    movel([0.140497, -1.371488, -2.576513, -0.764389, 1.570796, 1.711294],accel_mss,speed_ms,0,blend_radius_m)
    movel([0.140657, -1.371181, -2.576725, -0.764483, 1.570796, 1.711454],accel_mss,speed_ms,0,blend_radius_m)
    movel([0.140844, -1.370889, -2.576927, -0.764572, 1.570796, 1.711640],accel_mss,speed_ms,0,blend_radius_m)
    movel([0.141059, -1.370603, -2.577125, -0.764661, 1.570796, 1.711855],accel_mss,speed_ms,0,blend_radius_m)
    movel([0.141302, -1.370327, -2.577316, -0.764746, 1.570796, 1.712098],accel_mss,speed_ms,0,blend_radius_m)
    movel([0.141561, -1.370068, -2.577495, -0.764826, 1.570796, 1.712357],accel_mss,speed_ms,0,blend_radius_m)
    movel([0.141844, -1.369824, -2.577664, -0.764901, 1.570796, 1.712640],accel_mss,speed_ms,0,blend_radius_m)
    movel([0.142141, -1.369603, -2.577817, -0.764969, 1.570796, 1.712937],accel_mss,speed_ms,0,blend_radius_m)
    movel([0.142479, -1.369380, -2.577971, -0.765038, 1.570796, 1.713275],accel_mss,speed_ms,0,blend_radius_m)
    movel([0.142834, -1.369176, -2.578112, -0.765102, 1.570796, 1.713630],accel_mss,speed_ms,0,blend_radius_m)
    movel([0.143191, -1.368999, -2.578233, -0.765156, 1.570796, 1.713987],accel_mss,speed_ms,0,blend_radius_m)
    movel([0.143557, -1.368846, -2.578339, -0.765204, 1.570796, 1.714353],accel_mss,speed_ms,0,blend_radius_m)
    movel([0.143920, -1.368724, -2.578423, -0.765242, 1.570796, 1.714717],accel_mss,speed_ms,0,blend_radius_m)
    movel([0.144279, -1.368628, -2.578489, -0.765272, 1.570796, 1.715076],accel_mss,speed_ms,0,blend_radius_m)
    movel([0.144633, -1.368564, -2.578533, -0.765292, 1.570796, 1.715430],accel_mss,speed_ms,0,blend_radius_m)
    movel([0.144980, -1.368530, -2.578557, -0.765302, 1.570796, 1.715776],accel_mss,speed_ms,0,blend_radius_m)
    movel([0.145312, -1.368525, -2.578561, -0.765304, 1.570796, 1.716108],accel_mss,speed_ms,0,blend_radius_m)
    movel([0.145619, -1.368551, -2.578542, -0.765296, 1.570796, 1.716416],accel_mss,speed_ms,0,blend_radius_m)
    movel([0.145910, -1.368604, -2.578506, -0.765279, 1.570796, 1.716707],accel_mss,speed_ms,0,blend_radius_m)
    movel([0.146159, -1.368679, -2.578454, -0.765256, 1.570796, 1.716955],accel_mss,speed_ms,0,blend_radius_m)
    movel([0.146381, -1.368783, -2.578382, -0.765223, 1.570796, 1.717177],accel_mss,speed_ms,0,blend_radius_m)
    movel([0.146581, -1.368916, -2.578291, -0.765182, 1.570796, 1.717377],accel_mss,speed_ms,0,blend_radius_m)
    movel([0.146755, -1.369074, -2.578182, -0.765133, 1.570796, 1.717551],accel_mss,speed_ms,0,blend_radius_m)
    movel([0.146898, -1.369260, -2.578054, -0.765076, 1.570796, 1.717694],accel_mss,speed_ms,0,blend_radius_m)
    movel([0.147008, -1.369466, -2.577911, -0.765012, 1.570796, 1.717805],accel_mss,speed_ms,0,blend_radius_m)
    movel([0.147132, -1.369810, -2.577674, -0.764905, 1.570796, 1.717928],accel_mss,speed_ms,0,blend_radius_m)
    movel([0.147248, -1.370196, -2.577407, -0.764786, 1.570796, 1.718044],accel_mss,speed_ms,0,blend_radius_m)
    movel([0.147260, -1.370511, -2.577189, -0.764689, 1.570796, 1.718057],accel_mss,speed_ms,0,blend_radius_m)
    movel([0.147149, -1.370874, -2.576938, -0.764577, 1.570796, 1.717945],accel_mss,speed_ms,0,blend_radius_m)
    movel([0.146700, -1.371702, -2.576364, -0.764323, 1.570796, 1.717496],accel_mss,speed_ms,0,blend_radius_m)
    movel([0.146700, -1.374505, -2.577635, -0.760249, 1.570796, 1.717496],accel_mss,speed_ms,0,blend_radius_m)
    movel([0.146515, -1.374803, -2.577427, -0.760159, 1.570796, 1.717312],accel_mss,speed_ms,0,blend_radius_m)
    movel([0.146310, -1.375097, -2.577222, -0.760070, 1.570796, 1.717106],accel_mss,speed_ms,0,blend_radius_m)
    movel([0.146072, -1.375395, -2.577014, -0.759980, 1.570796, 1.716868],accel_mss,speed_ms,0,blend_radius_m)
    movel([0.145854, -1.375635, -2.576846, -0.759907, 1.570796, 1.716651],accel_mss,speed_ms,0,blend_radius_m)
    movel([0.145623, -1.375855, -2.576693, -0.759841, 1.570796, 1.716419],accel_mss,speed_ms,0,blend_radius_m)
    movel([0.145375, -1.376060, -2.576550, -0.759779, 1.570796, 1.716171],accel_mss,speed_ms,0,blend_radius_m)
    movel([0.145105, -1.376251, -2.576416, -0.759722, 1.570796, 1.715901],accel_mss,speed_ms,0,blend_radius_m)
    movel([0.144824, -1.376424, -2.576295, -0.759670, 1.570796, 1.715620],accel_mss,speed_ms,0,blend_radius_m)
    movel([0.144503, -1.376590, -2.576180, -0.759620, 1.570796, 1.715300],accel_mss,speed_ms,0,blend_radius_m)
    movel([0.144154, -1.376739, -2.576075, -0.759575, 1.570796, 1.714951],accel_mss,speed_ms,0,blend_radius_m)
    movel([0.143741, -1.376887, -2.575972, -0.759531, 1.570796, 1.714537],accel_mss,speed_ms,0,blend_radius_m)
    movel([0.143329, -1.377009, -2.575886, -0.759494, 1.570796, 1.714125],accel_mss,speed_ms,0,blend_radius_m)
    movel([0.142981, -1.377092, -2.575828, -0.759469, 1.570796, 1.713778],accel_mss,speed_ms,0,blend_radius_m)
    movel([0.142643, -1.377148, -2.575789, -0.759452, 1.570796, 1.713439],accel_mss,speed_ms,0,blend_radius_m)
    movel([0.142311, -1.377177, -2.575769, -0.759444, 1.570796, 1.713108],accel_mss,speed_ms,0,blend_radius_m)
    movel([0.141991, -1.377179, -2.575767, -0.759443, 1.570796, 1.712788],accel_mss,speed_ms,0,blend_radius_m)
    movel([0.141699, -1.377158, -2.575782, -0.759449, 1.570796, 1.712495],accel_mss,speed_ms,0,blend_radius_m)
    movel([0.141435, -1.377113, -2.575813, -0.759463, 1.570796, 1.712231],accel_mss,speed_ms,0,blend_radius_m)
    movel([0.141198, -1.377045, -2.575861, -0.759483, 1.570796, 1.711994],accel_mss,speed_ms,0,blend_radius_m)
    movel([0.140980, -1.376950, -2.575927, -0.759512, 1.570796, 1.711776],accel_mss,speed_ms,0,blend_radius_m)
    movel([0.140781, -1.376828, -2.576013, -0.759548, 1.570796, 1.711577],accel_mss,speed_ms,0,blend_radius_m)
    movel([0.140605, -1.376681, -2.576115, -0.759592, 1.570796, 1.711401],accel_mss,speed_ms,0,blend_radius_m)
    movel([0.140456, -1.376512, -2.576233, -0.759643, 1.570796, 1.711253],accel_mss,speed_ms,0,blend_radius_m)
    movel([0.140339, -1.376327, -2.576363, -0.759699, 1.570796, 1.711135],accel_mss,speed_ms,0,blend_radius_m)
    movel([0.140254, -1.376124, -2.576505, -0.759760, 1.570796, 1.711050],accel_mss,speed_ms,0,blend_radius_m)
    movel([0.140198, -1.375902, -2.576660, -0.759827, 1.570796, 1.710994],accel_mss,speed_ms,0,blend_radius_m)
    movel([0.140172, -1.375669, -2.576823, -0.759897, 1.570796, 1.710969],accel_mss,speed_ms,0,blend_radius_m)
    movel([0.140176, -1.375422, -2.576995, -0.759972, 1.570796, 1.710972],accel_mss,speed_ms,0,blend_radius_m)
    movel([0.140213, -1.375145, -2.577188, -0.760055, 1.570796, 1.711009],accel_mss,speed_ms,0,blend_radius_m)
    movel([0.140277, -1.374866, -2.577383, -0.760140, 1.570796, 1.711073],accel_mss,speed_ms,0,blend_radius_m)
    movel([0.140374, -1.374578, -2.577583, -0.760227, 1.570796, 1.711170],accel_mss,speed_ms,0,blend_radius_m)
    movel([0.140497, -1.374290, -2.577784, -0.760315, 1.570796, 1.711294],accel_mss,speed_ms,0,blend_radius_m)
    movel([0.140657, -1.373985, -2.577997, -0.760407, 1.570796, 1.711454],accel_mss,speed_ms,0,blend_radius_m)
    movel([0.140844, -1.373694, -2.578199, -0.760496, 1.570796, 1.711640],accel_mss,speed_ms,0,blend_radius_m)
    movel([0.141059, -1.373408, -2.578398, -0.760583, 1.570796, 1.711855],accel_mss,speed_ms,0,blend_radius_m)
    movel([0.141302, -1.373132, -2.578589, -0.760667, 1.570796, 1.712098],accel_mss,speed_ms,0,blend_radius_m)
    movel([0.141561, -1.372874, -2.578769, -0.760746, 1.570796, 1.712357],accel_mss,speed_ms,0,blend_radius_m)
    movel([0.141844, -1.372631, -2.578938, -0.760821, 1.570796, 1.712640],accel_mss,speed_ms,0,blend_radius_m)
    movel([0.142141, -1.372410, -2.579091, -0.760888, 1.570796, 1.712937],accel_mss,speed_ms,0,blend_radius_m)
    movel([0.142479, -1.372187, -2.579245, -0.760957, 1.570796, 1.713275],accel_mss,speed_ms,0,blend_radius_m)
    movel([0.142834, -1.371984, -2.579386, -0.761019, 1.570796, 1.713630],accel_mss,speed_ms,0,blend_radius_m)
    movel([0.143191, -1.371807, -2.579508, -0.761073, 1.570796, 1.713987],accel_mss,speed_ms,0,blend_radius_m)
    movel([0.143557, -1.371655, -2.579614, -0.761120, 1.570796, 1.714353],accel_mss,speed_ms,0,blend_radius_m)
    movel([0.143920, -1.371533, -2.579699, -0.761158, 1.570796, 1.714717],accel_mss,speed_ms,0,blend_radius_m)
    movel([0.144279, -1.371437, -2.579765, -0.761187, 1.570796, 1.715076],accel_mss,speed_ms,0,blend_radius_m)
    movel([0.144633, -1.371373, -2.579809, -0.761207, 1.570796, 1.715430],accel_mss,speed_ms,0,blend_radius_m)
    movel([0.144980, -1.371339, -2.579833, -0.761217, 1.570796, 1.715776],accel_mss,speed_ms,0,blend_radius_m)
    movel([0.145312, -1.371334, -2.579836, -0.761219, 1.570796, 1.716108],accel_mss,speed_ms,0,blend_radius_m)
    movel([0.145619, -1.371361, -2.579818, -0.761211, 1.570796, 1.716416],accel_mss,speed_ms,0,blend_radius_m)
    movel([0.145910, -1.371413, -2.579782, -0.761195, 1.570796, 1.716707],accel_mss,speed_ms,0,blend_radius_m)
    movel([0.146159, -1.371489, -2.579729, -0.761171, 1.570796, 1.716955],accel_mss,speed_ms,0,blend_radius_m)
    movel([0.146381, -1.371592, -2.579658, -0.761139, 1.570796, 1.717177],accel_mss,speed_ms,0,blend_radius_m)
    movel([0.146581, -1.371724, -2.579566, -0.761099, 1.570796, 1.717377],accel_mss,speed_ms,0,blend_radius_m)
    movel([0.146755, -1.371882, -2.579456, -0.761050, 1.570796, 1.717551],accel_mss,speed_ms,0,blend_radius_m)
    movel([0.146898, -1.372067, -2.579328, -0.760993, 1.570796, 1.717694],accel_mss,speed_ms,0,blend_radius_m)
    movel([0.147008, -1.372273, -2.579186, -0.760930, 1.570796, 1.717805],accel_mss,speed_ms,0,blend_radius_m)
    movel([0.147132, -1.372616, -2.578948, -0.760825, 1.570796, 1.717928],accel_mss,speed_ms,0,blend_radius_m)
    movel([0.147248, -1.373001, -2.578680, -0.760707, 1.570796, 1.718044],accel_mss,speed_ms,0,blend_radius_m)
    movel([0.147260, -1.373316, -2.578462, -0.760611, 1.570796, 1.718057],accel_mss,speed_ms,0,blend_radius_m)
    movel([0.147149, -1.373678, -2.578210, -0.760501, 1.570796, 1.717945],accel_mss,speed_ms,0,blend_radius_m)
    movel([0.146700, -1.374505, -2.577635, -0.760249, 1.570796, 1.717496],accel_mss,speed_ms,0,blend_radius_m)
    movel([0.146700, -1.341961, -2.561990, -0.808439, 1.570796, 1.717496],accel_mss,speed_ms,0,blend_radius_m)
    speed_ms = 1.000
    movel([0.156390, -1.339995, -2.563292, -0.809102, 1.570796, 1.727187],accel_mss,speed_ms,0,blend_radius_m)
    speed_ms = 0.008
    movel([0.156390, -1.366441, -2.576163, -0.769785, 1.570796, 1.727187],accel_mss,speed_ms,0,blend_radius_m)
    speed_ms = 0.003
    movel([0.156390, -1.369779, -2.577695, -0.764915, 1.570796, 1.727187],accel_mss,speed_ms,0,blend_radius_m)
    speed_ms = 0.008
    movel([0.155185, -1.370065, -2.577497, -0.764827, 1.570796, 1.725981],accel_mss,speed_ms,0,blend_radius_m)
    movel([0.156709, -1.361432, -2.583412, -0.767545, 1.570796, 1.727505],accel_mss,speed_ms,0,blend_radius_m)
    movel([0.159145, -1.360847, -2.583810, -0.767733, 1.570796, 1.729942],accel_mss,speed_ms,0,blend_radius_m)
    movel([0.157596, -1.369493, -2.577893, -0.765003, 1.570796, 1.728393],accel_mss,speed_ms,0,blend_radius_m)
    movel([0.156390, -1.369779, -2.577695, -0.764915, 1.570796, 1.727187],accel_mss,speed_ms,0,blend_radius_m)
    movel([0.156390, -1.372585, -2.578969, -0.760835, 1.570796, 1.727187],accel_mss,speed_ms,0,blend_radius_m)
    movel([0.155185, -1.372871, -2.578771, -0.760747, 1.570796, 1.725981],accel_mss,speed_ms,0,blend_radius_m)
    movel([0.156709, -1.364257, -2.584698, -0.763434, 1.570796, 1.727505],accel_mss,speed_ms,0,blend_radius_m)
    movel([0.159145, -1.363673, -2.585096, -0.763620, 1.570796, 1.729942],accel_mss,speed_ms,0,blend_radius_m)
    movel([0.157596, -1.372300, -2.579167, -0.760922, 1.570796, 1.728393],accel_mss,speed_ms,0,blend_radius_m)
    movel([0.156390, -1.372585, -2.578969, -0.760835, 1.570796, 1.727187],accel_mss,speed_ms,0,blend_radius_m)
    movel([0.156390, -1.339995, -2.563292, -0.809102, 1.570796, 1.727187],accel_mss,speed_ms,0,blend_radius_m)
    speed_ms = 1.000
    movel([0.133729, -1.353431, -2.554289, -0.804669, 1.570796, 1.704526],accel_mss,speed_ms,0,blend_radius_m)
    speed_ms = 0.008
    movel([0.133729, -1.379621, -2.566981, -0.765787, 1.570796, 1.704526],accel_mss,speed_ms,0,blend_radius_m)
    speed_ms = 0.003
    movel([0.133729, -1.382923, -2.568492, -0.760974, 1.570796, 1.704526],accel_mss,speed_ms,0,blend_radius_m)
    speed_ms = 0.008
    movel([0.114781, -1.387789, -2.565022, -0.759578, 1.570796, 1.685577],accel_mss,speed_ms,0,blend_radius_m)
    movel([0.118930, -1.356883, -2.586487, -0.769019, 1.570796, 1.689727],accel_mss,speed_ms,0,blend_radius_m)
    movel([0.158436, -1.346557, -2.593359, -0.772473, 1.570796, 1.729232],accel_mss,speed_ms,0,blend_radius_m)
    movel([0.152738, -1.378302, -2.571755, -0.762332, 1.570796, 1.723534],accel_mss,speed_ms,0,blend_radius_m)
    movel([0.133729, -1.382923, -2.568492, -0.760974, 1.570796, 1.704526],accel_mss,speed_ms,0,blend_radius_m)
    movel([0.133729, -1.385699, -2.569747, -0.756942, 1.570796, 1.704526],accel_mss,speed_ms,0,blend_radius_m)
    movel([0.114781, -1.390554, -2.566271, -0.755564, 1.570796, 1.685577],accel_mss,speed_ms,0,blend_radius_m)
    movel([0.118930, -1.359718, -2.587779, -0.764892, 1.570796, 1.689727],accel_mss,speed_ms,0,blend_radius_m)
    movel([0.158436, -1.349414, -2.594666, -0.768309, 1.570796, 1.729232],accel_mss,speed_ms,0,blend_radius_m)
    movel([0.152738, -1.381089, -2.573017, -0.758282, 1.570796, 1.723534],accel_mss,speed_ms,0,blend_radius_m)
    movel([0.133729, -1.385699, -2.569747, -0.756942, 1.570796, 1.704526],accel_mss,speed_ms,0,blend_radius_m)
    movel([0.133729, -1.353431, -2.554289, -0.804669, 1.570796, 1.704526],accel_mss,speed_ms,0,blend_radius_m)
    speed_ms = 1.000
    movel([0.133180, -1.357101, -2.551788, -0.803501, 1.570796, 1.703976],accel_mss,speed_ms,0,blend_radius_m)
    speed_ms = 0.008
    movel([0.133180, -1.383219, -2.564431, -0.764739, 1.570796, 1.703976],accel_mss,speed_ms,0,blend_radius_m)
    speed_ms = 0.003
    movel([0.133180, -1.386511, -2.565936, -0.759942, 1.570796, 1.703976],accel_mss,speed_ms,0,blend_radius_m)
    speed_ms = 0.008
    movel([0.125117, -1.388474, -2.564530, -0.759385, 1.570796, 1.695913],accel_mss,speed_ms,0,blend_radius_m)
    movel([0.125288, -1.386059, -2.566259, -0.760071, 1.570796, 1.696085],accel_mss,speed_ms,0,blend_radius_m)
    movel([0.141678, -1.381967, -2.569169, -0.761253, 1.570796, 1.712474],accel_mss,speed_ms,0,blend_radius_m)
    movel([0.141253, -1.384594, -2.567304, -0.760491, 1.570796, 1.712049],accel_mss,speed_ms,0,blend_radius_m)
    movel([0.133180, -1.386511, -2.565936, -0.759942, 1.570796, 1.703976],accel_mss,speed_ms,0,blend_radius_m)
    movel([0.133180, -1.389280, -2.567187, -0.755923, 1.570796, 1.703976],accel_mss,speed_ms,0,blend_radius_m)
    movel([0.125117, -1.391238, -2.565778, -0.755373, 1.570796, 1.695913],accel_mss,speed_ms,0,blend_radius_m)
    movel([0.125288, -1.388829, -2.567510, -0.756050, 1.570796, 1.696085],accel_mss,speed_ms,0,blend_radius_m)
    movel([0.141678, -1.384746, -2.570426, -0.757217, 1.570796, 1.712474],accel_mss,speed_ms,0,blend_radius_m)
    movel([0.141253, -1.387367, -2.568557, -0.756465, 1.570796, 1.712049],accel_mss,speed_ms,0,blend_radius_m)
    movel([0.133180, -1.389280, -2.567187, -0.755923, 1.570796, 1.703976],accel_mss,speed_ms,0,blend_radius_m)
    movel([0.133180, -1.357101, -2.551788, -0.803501, 1.570796, 1.703976],accel_mss,speed_ms,0,blend_radius_m)
    speed_ms = 1.000
    movel([0.128927, -1.347517, -2.558282, -0.806591, 1.570796, 1.699723],accel_mss,speed_ms,0,blend_radius_m)
    speed_ms = 0.008
    movel([0.128927, -1.373820, -2.571052, -0.767516, 1.570796, 1.699723],accel_mss,speed_ms,0,blend_radius_m)
    speed_ms = 0.003
    movel([0.128927, -1.377138, -2.572573, -0.762678, 1.570796, 1.699723],accel_mss,speed_ms,0,blend_radius_m)
    speed_ms = 0.008
    movel([0.128678, -1.377358, -2.572418, -0.762613, 1.570796, 1.699474],accel_mss,speed_ms,0,blend_radius_m)
    movel([0.128417, -1.377567, -2.572272, -0.762550, 1.570796, 1.699213],accel_mss,speed_ms,0,blend_radius_m)
    movel([0.128143, -1.377759, -2.572137, -0.762493, 1.570796, 1.698939],accel_mss,speed_ms,0,blend_radius_m)
    movel([0.127865, -1.377934, -2.572014, -0.762441, 1.570796, 1.698661],accel_mss,speed_ms,0,blend_radius_m)
    movel([0.127577, -1.378092, -2.571903, -0.762394, 1.570796, 1.698374],accel_mss,speed_ms,0,blend_radius_m)
    movel([0.127288, -1.378230, -2.571806, -0.762353, 1.570796, 1.698084],accel_mss,speed_ms,0,blend_radius_m)
    movel([0.126992, -1.378351, -2.571721, -0.762317, 1.570796, 1.697788],accel_mss,speed_ms,0,blend_radius_m)
    movel([0.126696, -1.378450, -2.571651, -0.762288, 1.570796, 1.697492],accel_mss,speed_ms,0,blend_radius_m)
    movel([0.126398, -1.378531, -2.571594, -0.762263, 1.570796, 1.697195],accel_mss,speed_ms,0,blend_radius_m)
    movel([0.126104, -1.378591, -2.571552, -0.762246, 1.570796, 1.696900],accel_mss,speed_ms,0,blend_radius_m)
    movel([0.125815, -1.378625, -2.571528, -0.762236, 1.570796, 1.696611],accel_mss,speed_ms,0,blend_radius_m)
    movel([0.125536, -1.378641, -2.571517, -0.762231, 1.570796, 1.696333],accel_mss,speed_ms,0,blend_radius_m)
    movel([0.125266, -1.378631, -2.571524, -0.762234, 1.570796, 1.696063],accel_mss,speed_ms,0,blend_radius_m)
    movel([0.125011, -1.378600, -2.571546, -0.762243, 1.570796, 1.695807],accel_mss,speed_ms,0,blend_radius_m)
    movel([0.124771, -1.378546, -2.571584, -0.762259, 1.570796, 1.695567],accel_mss,speed_ms,0,blend_radius_m)
    movel([0.124546, -1.378470, -2.571637, -0.762282, 1.570796, 1.695343],accel_mss,speed_ms,0,blend_radius_m)
    movel([0.124337, -1.378373, -2.571705, -0.762310, 1.570796, 1.695133],accel_mss,speed_ms,0,blend_radius_m)
    movel([0.124147, -1.378252, -2.571791, -0.762346, 1.570796, 1.694943],accel_mss,speed_ms,0,blend_radius_m)
    movel([0.123977, -1.378113, -2.571888, -0.762388, 1.570796, 1.694773],accel_mss,speed_ms,0,blend_radius_m)
    movel([0.123831, -1.377953, -2.572001, -0.762435, 1.570796, 1.694627],accel_mss,speed_ms,0,blend_radius_m)
    movel([0.123713, -1.377783, -2.572120, -0.762486, 1.570796, 1.694510],accel_mss,speed_ms,0,blend_radius_m)
    movel([0.123619, -1.377597, -2.572250, -0.762541, 1.570796, 1.694416],accel_mss,speed_ms,0,blend_radius_m)
    movel([0.123552, -1.377393, -2.572393, -0.762602, 1.570796, 1.694348],accel_mss,speed_ms,0,blend_radius_m)
    movel([0.123508, -1.377177, -2.572545, -0.762667, 1.570796, 1.694304],accel_mss,speed_ms,0,blend_radius_m)
    movel([0.123493, -1.376928, -2.572720, -0.762741, 1.570796, 1.694289],accel_mss,speed_ms,0,blend_radius_m)
    movel([0.123508, -1.376667, -2.572903, -0.762819, 1.570796, 1.694304],accel_mss,speed_ms,0,blend_radius_m)
    movel([0.123557, -1.376371, -2.573110, -0.762908, 1.570796, 1.694353],accel_mss,speed_ms,0,blend_radius_m)
    movel([0.123637, -1.376065, -2.573324, -0.763000, 1.570796, 1.694433],accel_mss,speed_ms,0,blend_radius_m)
    movel([0.123817, -1.375642, -2.573621, -0.763127, 1.570796, 1.694614],accel_mss,speed_ms,0,blend_radius_m)
    movel([0.124117, -1.375197, -2.573931, -0.763261, 1.570796, 1.694913],accel_mss,speed_ms,0,blend_radius_m)
    movel([0.124404, -1.374864, -2.574164, -0.763361, 1.570796, 1.695200],accel_mss,speed_ms,0,blend_radius_m)
    movel([0.124768, -1.374474, -2.574436, -0.763479, 1.570796, 1.695565],accel_mss,speed_ms,0,blend_radius_m)
    movel([0.125177, -1.374069, -2.574718, -0.763602, 1.570796, 1.695973],accel_mss,speed_ms,0,blend_radius_m)
    movel([0.125601, -1.373672, -2.574995, -0.763722, 1.570796, 1.696398],accel_mss,speed_ms,0,blend_radius_m)
    movel([0.125949, -1.373409, -2.575178, -0.763802, 1.570796, 1.696745],accel_mss,speed_ms,0,blend_radius_m)
    movel([0.126328, -1.373213, -2.575315, -0.763862, 1.570796, 1.697124],accel_mss,speed_ms,0,blend_radius_m)
    movel([0.126597, -1.373121, -2.575378, -0.763890, 1.570796, 1.697393],accel_mss,speed_ms,0,blend_radius_m)
    movel([0.127212, -1.372982, -2.575475, -0.763932, 1.570796, 1.698008],accel_mss,speed_ms,0,blend_radius_m)
    movel([0.127706, -1.372894, -2.575536, -0.763959, 1.570796, 1.698502],accel_mss,speed_ms,0,blend_radius_m)
    movel([0.128139, -1.372845, -2.575570, -0.763974, 1.570796, 1.698935],accel_mss,speed_ms,0,blend_radius_m)
    movel([0.128566, -1.372832, -2.575579, -0.763978, 1.570796, 1.699362],accel_mss,speed_ms,0,blend_radius_m)
    movel([0.128976, -1.372853, -2.575565, -0.763971, 1.570796, 1.699773],accel_mss,speed_ms,0,blend_radius_m)
    movel([0.129257, -1.372899, -2.575532, -0.763957, 1.570796, 1.700053],accel_mss,speed_ms,0,blend_radius_m)
    movel([0.129513, -1.372980, -2.575477, -0.763933, 1.570796, 1.700310],accel_mss,speed_ms,0,blend_radius_m)
    movel([0.129747, -1.373100, -2.575393, -0.763896, 1.570796, 1.700543],accel_mss,speed_ms,0,blend_radius_m)
    movel([0.129949, -1.373251, -2.575288, -0.763850, 1.570796, 1.700745],accel_mss,speed_ms,0,blend_radius_m)
    movel([0.130106, -1.373427, -2.575165, -0.763796, 1.570796, 1.700903],accel_mss,speed_ms,0,blend_radius_m)
    movel([0.130226, -1.373632, -2.575023, -0.763734, 1.570796, 1.701022],accel_mss,speed_ms,0,blend_radius_m)
    movel([0.130303, -1.373860, -2.574864, -0.763665, 1.570796, 1.701099],accel_mss,speed_ms,0,blend_radius_m)
    movel([0.130342, -1.374113, -2.574687, -0.763588, 1.570796, 1.701138],accel_mss,speed_ms,0,blend_radius_m)
    movel([0.130351, -1.374427, -2.574469, -0.763493, 1.570796, 1.701147],accel_mss,speed_ms,0,blend_radius_m)
    movel([0.130321, -1.374754, -2.574240, -0.763394, 1.570796, 1.701117],accel_mss,speed_ms,0,blend_radius_m)
    movel([0.130262, -1.375070, -2.574020, -0.763299, 1.570796, 1.701058],accel_mss,speed_ms,0,blend_radius_m)
    movel([0.130173, -1.375375, -2.573807, -0.763207, 1.570796, 1.700970],accel_mss,speed_ms,0,blend_radius_m)
    movel([0.130057, -1.375652, -2.573613, -0.763124, 1.570796, 1.700854],accel_mss,speed_ms,0,blend_radius_m)
    movel([0.129902, -1.375947, -2.573407, -0.763035, 1.570796, 1.700699],accel_mss,speed_ms,0,blend_radius_m)
    movel([0.129708, -1.376249, -2.573196, -0.762944, 1.570796, 1.700505],accel_mss,speed_ms,0,blend_radius_m)
    movel([0.129478, -1.376551, -2.572984, -0.762854, 1.570796, 1.700275],accel_mss,speed_ms,0,blend_radius_m)
    movel([0.129215, -1.376849, -2.572776, -0.762765, 1.570796, 1.700012],accel_mss,speed_ms,0,blend_radius_m)
    movel([0.128927, -1.377138, -2.572573, -0.762678, 1.570796, 1.699723],accel_mss,speed_ms,0,blend_radius_m)
    movel([0.128927, -1.379928, -2.573836, -0.758625, 1.570796, 1.699723],accel_mss,speed_ms,0,blend_radius_m)
    movel([0.128678, -1.380147, -2.573682, -0.758560, 1.570796, 1.699474],accel_mss,speed_ms,0,blend_radius_m)
    movel([0.128417, -1.380356, -2.573535, -0.758498, 1.570796, 1.699213],accel_mss,speed_ms,0,blend_radius_m)
    movel([0.128143, -1.380548, -2.573399, -0.758442, 1.570796, 1.698939],accel_mss,speed_ms,0,blend_radius_m)
    movel([0.127865, -1.380722, -2.573276, -0.758390, 1.570796, 1.698661],accel_mss,speed_ms,0,blend_radius_m)
    movel([0.127577, -1.380880, -2.573165, -0.758344, 1.570796, 1.698374],accel_mss,speed_ms,0,blend_radius_m)
    movel([0.127288, -1.381018, -2.573068, -0.758303, 1.570796, 1.698084],accel_mss,speed_ms,0,blend_radius_m)
    movel([0.126992, -1.381138, -2.572983, -0.758268, 1.570796, 1.697788],accel_mss,speed_ms,0,blend_radius_m)
    movel([0.126696, -1.381237, -2.572913, -0.758239, 1.570796, 1.697492],accel_mss,speed_ms,0,blend_radius_m)
    movel([0.126398, -1.381318, -2.572856, -0.758215, 1.570796, 1.697195],accel_mss,speed_ms,0,blend_radius_m)
    movel([0.126104, -1.381377, -2.572814, -0.758198, 1.570796, 1.696900],accel_mss,speed_ms,0,blend_radius_m)
    movel([0.125815, -1.381412, -2.572790, -0.758188, 1.570796, 1.696611],accel_mss,speed_ms,0,blend_radius_m)
    movel([0.125536, -1.381427, -2.572779, -0.758183, 1.570796, 1.696333],accel_mss,speed_ms,0,blend_radius_m)
    movel([0.125266, -1.381417, -2.572786, -0.758186, 1.570796, 1.696063],accel_mss,speed_ms,0,blend_radius_m)
    movel([0.125011, -1.381387, -2.572807, -0.758195, 1.570796, 1.695807],accel_mss,speed_ms,0,blend_radius_m)
    movel([0.124771, -1.381333, -2.572845, -0.758211, 1.570796, 1.695567],accel_mss,speed_ms,0,blend_radius_m)
    movel([0.124546, -1.381257, -2.572899, -0.758233, 1.570796, 1.695343],accel_mss,speed_ms,0,blend_radius_m)
    movel([0.124337, -1.381160, -2.572967, -0.758261, 1.570796, 1.695133],accel_mss,speed_ms,0,blend_radius_m)
    movel([0.124147, -1.381039, -2.573053, -0.758297, 1.570796, 1.694943],accel_mss,speed_ms,0,blend_radius_m)
    movel([0.123977, -1.380901, -2.573151, -0.758338, 1.570796, 1.694773],accel_mss,speed_ms,0,blend_radius_m)
    movel([0.123831, -1.380741, -2.573263, -0.758385, 1.570796, 1.694627],accel_mss,speed_ms,0,blend_radius_m)
    movel([0.123713, -1.380572, -2.573382, -0.758435, 1.570796, 1.694510],accel_mss,speed_ms,0,blend_radius_m)
    movel([0.123619, -1.380386, -2.573513, -0.758489, 1.570796, 1.694416],accel_mss,speed_ms,0,blend_radius_m)
    movel([0.123552, -1.380183, -2.573657, -0.758549, 1.570796, 1.694348],accel_mss,speed_ms,0,blend_radius_m)
    movel([0.123508, -1.379967, -2.573809, -0.758613, 1.570796, 1.694304],accel_mss,speed_ms,0,blend_radius_m)
    movel([0.123493, -1.379719, -2.573984, -0.758687, 1.570796, 1.694289],accel_mss,speed_ms,0,blend_radius_m)
    movel([0.123508, -1.379458, -2.574167, -0.758764, 1.570796, 1.694304],accel_mss,speed_ms,0,blend_radius_m)
    movel([0.123557, -1.379163, -2.574375, -0.758851, 1.570796, 1.694353],accel_mss,speed_ms,0,blend_radius_m)
    movel([0.123637, -1.378857, -2.574589, -0.758942, 1.570796, 1.694433],accel_mss,speed_ms,0,blend_radius_m)
    movel([0.123817, -1.378435, -2.574886, -0.759068, 1.570796, 1.694614],accel_mss,speed_ms,0,blend_radius_m)
    movel([0.124117, -1.377992, -2.575197, -0.759200, 1.570796, 1.694913],accel_mss,speed_ms,0,blend_radius_m)
    movel([0.124404, -1.377659, -2.575430, -0.759299, 1.570796, 1.695200],accel_mss,speed_ms,0,blend_radius_m)
    movel([0.124768, -1.377270, -2.575703, -0.759416, 1.570796, 1.695565],accel_mss,speed_ms,0,blend_radius_m)
    movel([0.125177, -1.376866, -2.575986, -0.759537, 1.570796, 1.695973],accel_mss,speed_ms,0,blend_radius_m)
    movel([0.125601, -1.376470, -2.576263, -0.759656, 1.570796, 1.696398],accel_mss,speed_ms,0,blend_radius_m)
    movel([0.125949, -1.376208, -2.576447, -0.759735, 1.570796, 1.696745],accel_mss,speed_ms,0,blend_radius_m)
    movel([0.126328, -1.376012, -2.576584, -0.759794, 1.570796, 1.697124],accel_mss,speed_ms,0,blend_radius_m)
    movel([0.126597, -1.375920, -2.576647, -0.759821, 1.570796, 1.697393],accel_mss,speed_ms,0,blend_radius_m)
    movel([0.127212, -1.375782, -2.576744, -0.759863, 1.570796, 1.698008],accel_mss,speed_ms,0,blend_radius_m)
    movel([0.127706, -1.375694, -2.576806, -0.759890, 1.570796, 1.698502],accel_mss,speed_ms,0,blend_radius_m)
    movel([0.128139, -1.375645, -2.576840, -0.759904, 1.570796, 1.698935],accel_mss,speed_ms,0,blend_radius_m)
    movel([0.128566, -1.375632, -2.576849, -0.759908, 1.570796, 1.699362],accel_mss,speed_ms,0,blend_radius_m)
    movel([0.128976, -1.375653, -2.576834, -0.759902, 1.570796, 1.699773],accel_mss,speed_ms,0,blend_radius_m)
    movel([0.129257, -1.375699, -2.576802, -0.759888, 1.570796, 1.700053],accel_mss,speed_ms,0,blend_radius_m)
    movel([0.129513, -1.375779, -2.576746, -0.759864, 1.570796, 1.700310],accel_mss,speed_ms,0,blend_radius_m)
    movel([0.129747, -1.375899, -2.576662, -0.759828, 1.570796, 1.700543],accel_mss,speed_ms,0,blend_radius_m)
    movel([0.129949, -1.376050, -2.576557, -0.759782, 1.570796, 1.700745],accel_mss,speed_ms,0,blend_radius_m)
    movel([0.130106, -1.376226, -2.576434, -0.759729, 1.570796, 1.700903],accel_mss,speed_ms,0,blend_radius_m)
    movel([0.130226, -1.376430, -2.576291, -0.759668, 1.570796, 1.701022],accel_mss,speed_ms,0,blend_radius_m)
    movel([0.130303, -1.376658, -2.576132, -0.759599, 1.570796, 1.701099],accel_mss,speed_ms,0,blend_radius_m)
    movel([0.130342, -1.376910, -2.575955, -0.759524, 1.570796, 1.701138],accel_mss,speed_ms,0,blend_radius_m)
    movel([0.130351, -1.377223, -2.575736, -0.759430, 1.570796, 1.701147],accel_mss,speed_ms,0,blend_radius_m)
    movel([0.130321, -1.377550, -2.575507, -0.759332, 1.570796, 1.701117],accel_mss,speed_ms,0,blend_radius_m)
    movel([0.130262, -1.377865, -2.575286, -0.759238, 1.570796, 1.701058],accel_mss,speed_ms,0,blend_radius_m)
    movel([0.130173, -1.378168, -2.575073, -0.759147, 1.570796, 1.700970],accel_mss,speed_ms,0,blend_radius_m)
    movel([0.130057, -1.378445, -2.574879, -0.759065, 1.570796, 1.700854],accel_mss,speed_ms,0,blend_radius_m)
    movel([0.129902, -1.378740, -2.574672, -0.758977, 1.570796, 1.700699],accel_mss,speed_ms,0,blend_radius_m)
    movel([0.129708, -1.379041, -2.574461, -0.758888, 1.570796, 1.700505],accel_mss,speed_ms,0,blend_radius_m)
    movel([0.129478, -1.379342, -2.574249, -0.758798, 1.570796, 1.700275],accel_mss,speed_ms,0,blend_radius_m)
    movel([0.129215, -1.379639, -2.574040, -0.758710, 1.570796, 1.700012],accel_mss,speed_ms,0,blend_radius_m)
    movel([0.128927, -1.379928, -2.573836, -0.758625, 1.570796, 1.699723],accel_mss,speed_ms,0,blend_radius_m)
    movel([0.128927, -1.347517, -2.558282, -0.806591, 1.570796, 1.699723],accel_mss,speed_ms,0,blend_radius_m)
    speed_ms = 1.000
    movel([0.129045, -1.344649, -2.560200, -0.807539, 1.570796, 1.699842],accel_mss,speed_ms,0,blend_radius_m)
    speed_ms = 0.008
    movel([0.129045, -1.371008, -2.573009, -0.768372, 1.570796, 1.699842],accel_mss,speed_ms,0,blend_radius_m)
    speed_ms = 0.003
    movel([0.129045, -1.374333, -2.574534, -0.763522, 1.570796, 1.699842],accel_mss,speed_ms,0,blend_radius_m)
    speed_ms = 0.008
    movel([0.128893, -1.374056, -2.574727, -0.763605, 1.570796, 1.699689],accel_mss,speed_ms,0,blend_radius_m)
    movel([0.128656, -1.373849, -2.574872, -0.763668, 1.570796, 1.699452],accel_mss,speed_ms,0,blend_radius_m)
    movel([0.128349, -1.373716, -2.574964, -0.763709, 1.570796, 1.699146],accel_mss,speed_ms,0,blend_radius_m)
    movel([0.127975, -1.373664, -2.575000, -0.763724, 1.570796, 1.698771],accel_mss,speed_ms,0,blend_radius_m)
    movel([0.127549, -1.373690, -2.574982, -0.763717, 1.570796, 1.698345],accel_mss,speed_ms,0,blend_radius_m)
    movel([0.127101, -1.373796, -2.574908, -0.763684, 1.570796, 1.697897],accel_mss,speed_ms,0,blend_radius_m)
    movel([0.126646, -1.373980, -2.574780, -0.763629, 1.570796, 1.697443],accel_mss,speed_ms,0,blend_radius_m)
    movel([0.126199, -1.374234, -2.574603, -0.763552, 1.570796, 1.696995],accel_mss,speed_ms,0,blend_radius_m)
    movel([0.125788, -1.374541, -2.574390, -0.763459, 1.570796, 1.696584],accel_mss,speed_ms,0,blend_radius_m)
    movel([0.125421, -1.374895, -2.574142, -0.763352, 1.570796, 1.696217],accel_mss,speed_ms,0,blend_radius_m)
    movel([0.125130, -1.375256, -2.573890, -0.763243, 1.570796, 1.695926],accel_mss,speed_ms,0,blend_radius_m)
    movel([0.124906, -1.375638, -2.573623, -0.763128, 1.570796, 1.695702],accel_mss,speed_ms,0,blend_radius_m)
    movel([0.124761, -1.376024, -2.573353, -0.763012, 1.570796, 1.695558],accel_mss,speed_ms,0,blend_radius_m)
    movel([0.124703, -1.376401, -2.573089, -0.762899, 1.570796, 1.695499],accel_mss,speed_ms,0,blend_radius_m)
    movel([0.124725, -1.376765, -2.572835, -0.762790, 1.570796, 1.695522],accel_mss,speed_ms,0,blend_radius_m)
    movel([0.124831, -1.377087, -2.572608, -0.762693, 1.570796, 1.695627],accel_mss,speed_ms,0,blend_radius_m)
    movel([0.125011, -1.377346, -2.572427, -0.762616, 1.570796, 1.695807],accel_mss,speed_ms,0,blend_radius_m)
    movel([0.125259, -1.377541, -2.572290, -0.762558, 1.570796, 1.696056],accel_mss,speed_ms,0,blend_radius_m)
    movel([0.125573, -1.377666, -2.572202, -0.762521, 1.570796, 1.696370],accel_mss,speed_ms,0,blend_radius_m)
    movel([0.125937, -1.377715, -2.572168, -0.762506, 1.570796, 1.696733],accel_mss,speed_ms,0,blend_radius_m)
    movel([0.126338, -1.377687, -2.572187, -0.762514, 1.570796, 1.697134],accel_mss,speed_ms,0,blend_radius_m)
    movel([0.126757, -1.377585, -2.572259, -0.762545, 1.570796, 1.697553],accel_mss,speed_ms,0,blend_radius_m)
    movel([0.127186, -1.377411, -2.572381, -0.762597, 1.570796, 1.697983],accel_mss,speed_ms,0,blend_radius_m)
    movel([0.127611, -1.377168, -2.572551, -0.762669, 1.570796, 1.698408],accel_mss,speed_ms,0,blend_radius_m)
    movel([0.128014, -1.376868, -2.572762, -0.762759, 1.570796, 1.698810],accel_mss,speed_ms,0,blend_radius_m)
    movel([0.128380, -1.376523, -2.573004, -0.762862, 1.570796, 1.699176],accel_mss,speed_ms,0,blend_radius_m)
    movel([0.128590, -1.376291, -2.573166, -0.762932, 1.570796, 1.699386],accel_mss,speed_ms,0,blend_radius_m)
    movel([0.128781, -1.376054, -2.573332, -0.763003, 1.570796, 1.699578],accel_mss,speed_ms,0,blend_radius_m)
    movel([0.129007, -1.375700, -2.573580, -0.763109, 1.570796, 1.699803],accel_mss,speed_ms,0,blend_radius_m)
    movel([0.129132, -1.375380, -2.573803, -0.763206, 1.570796, 1.699928],accel_mss,speed_ms,0,blend_radius_m)
    movel([0.129180, -1.375067, -2.574022, -0.763300, 1.570796, 1.699977],accel_mss,speed_ms,0,blend_radius_m)
    movel([0.129142, -1.374706, -2.574274, -0.763409, 1.570796, 1.699938],accel_mss,speed_ms,0,blend_radius_m)
    movel([0.129045, -1.374333, -2.574534, -0.763522, 1.570796, 1.699842],accel_mss,speed_ms,0,blend_radius_m)
    movel([0.129045, -1.377129, -2.575802, -0.759458, 1.570796, 1.699842],accel_mss,speed_ms,0,blend_radius_m)
    movel([0.128893, -1.376853, -2.575995, -0.759541, 1.570796, 1.699689],accel_mss,speed_ms,0,blend_radius_m)
    movel([0.128656, -1.376646, -2.576140, -0.759603, 1.570796, 1.699452],accel_mss,speed_ms,0,blend_radius_m)
    movel([0.128349, -1.376514, -2.576233, -0.759643, 1.570796, 1.699146],accel_mss,speed_ms,0,blend_radius_m)
    movel([0.127975, -1.376462, -2.576269, -0.759658, 1.570796, 1.698771],accel_mss,speed_ms,0,blend_radius_m)
    movel([0.127549, -1.376488, -2.576251, -0.759650, 1.570796, 1.698345],accel_mss,speed_ms,0,blend_radius_m)
    movel([0.127101, -1.376594, -2.576177, -0.759619, 1.570796, 1.697897],accel_mss,speed_ms,0,blend_radius_m)
    movel([0.126646, -1.376777, -2.576048, -0.759564, 1.570796, 1.697443],accel_mss,speed_ms,0,blend_radius_m)
    movel([0.126199, -1.377031, -2.575871, -0.759487, 1.570796, 1.696995],accel_mss,speed_ms,0,blend_radius_m)
    movel([0.125788, -1.377336, -2.575657, -0.759396, 1.570796, 1.696584],accel_mss,speed_ms,0,blend_radius_m)
    movel([0.125421, -1.377690, -2.575409, -0.759290, 1.570796, 1.696217],accel_mss,speed_ms,0,blend_radius_m)
    movel([0.125130, -1.378050, -2.575156, -0.759182, 1.570796, 1.695926],accel_mss,speed_ms,0,blend_radius_m)
    movel([0.124906, -1.378431, -2.574889, -0.759069, 1.570796, 1.695702],accel_mss,speed_ms,0,blend_radius_m)
    movel([0.124761, -1.378817, -2.574618, -0.758954, 1.570796, 1.695558],accel_mss,speed_ms,0,blend_radius_m)
    movel([0.124703, -1.379193, -2.574354, -0.758843, 1.570796, 1.695499],accel_mss,speed_ms,0,blend_radius_m)
    movel([0.124725, -1.379555, -2.574099, -0.758735, 1.570796, 1.695522],accel_mss,speed_ms,0,blend_radius_m)
    movel([0.124831, -1.379877, -2.573872, -0.758640, 1.570796, 1.695627],accel_mss,speed_ms,0,blend_radius_m)
    movel([0.125011, -1.380136, -2.573690, -0.758563, 1.570796, 1.695807],accel_mss,speed_ms,0,blend_radius_m)
    movel([0.125259, -1.380330, -2.573553, -0.758506, 1.570796, 1.696056],accel_mss,speed_ms,0,blend_radius_m)
    movel([0.125573, -1.380455, -2.573465, -0.758469, 1.570796, 1.696370],accel_mss,speed_ms,0,blend_radius_m)
    movel([0.125937, -1.380504, -2.573430, -0.758455, 1.570796, 1.696733],accel_mss,speed_ms,0,blend_radius_m)
    movel([0.126338, -1.380476, -2.573450, -0.758463, 1.570796, 1.697134],accel_mss,speed_ms,0,blend_radius_m)
    movel([0.126757, -1.380374, -2.573522, -0.758493, 1.570796, 1.697553],accel_mss,speed_ms,0,blend_radius_m)
    movel([0.127186, -1.380200, -2.573644, -0.758544, 1.570796, 1.697983],accel_mss,speed_ms,0,blend_radius_m)
    movel([0.127611, -1.379958, -2.573815, -0.758616, 1.570796, 1.698408],accel_mss,speed_ms,0,blend_radius_m)
    movel([0.128014, -1.379659, -2.574026, -0.758704, 1.570796, 1.698810],accel_mss,speed_ms,0,blend_radius_m)
    movel([0.128380, -1.379314, -2.574268, -0.758807, 1.570796, 1.699176],accel_mss,speed_ms,0,blend_radius_m)
    movel([0.128590, -1.379083, -2.574431, -0.758875, 1.570796, 1.699386],accel_mss,speed_ms,0,blend_radius_m)
    movel([0.128781, -1.378846, -2.574597, -0.758945, 1.570796, 1.699578],accel_mss,speed_ms,0,blend_radius_m)
    movel([0.129007, -1.378493, -2.574846, -0.759051, 1.570796, 1.699803],accel_mss,speed_ms,0,blend_radius_m)
    movel([0.129132, -1.378174, -2.575069, -0.759146, 1.570796, 1.699928],accel_mss,speed_ms,0,blend_radius_m)
    movel([0.129180, -1.377862, -2.575289, -0.759239, 1.570796, 1.699977],accel_mss,speed_ms,0,blend_radius_m)
    movel([0.129142, -1.377502, -2.575541, -0.759346, 1.570796, 1.699938],accel_mss,speed_ms,0,blend_radius_m)
    movel([0.129045, -1.377129, -2.575802, -0.759458, 1.570796, 1.699842],accel_mss,speed_ms,0,blend_radius_m)
    movel([0.129045, -1.344649, -2.560200, -0.807539, 1.570796, 1.699842],accel_mss,speed_ms,0,blend_radius_m)
    speed_ms = 1.000
    movel([0.131028, -1.343086, -2.561242, -0.808061, 1.570796, 1.701824],accel_mss,speed_ms,0,blend_radius_m)
    speed_ms = 0.008
    movel([0.131028, -1.369474, -2.574072, -0.768843, 1.570796, 1.701824],accel_mss,speed_ms,0,blend_radius_m)
    speed_ms = 0.003
    movel([0.131028, -1.372804, -2.575599, -0.763986, 1.570796, 1.701824],accel_mss,speed_ms,0,blend_radius_m)
    speed_ms = 0.008
    movel([0.130850, -1.372573, -2.575759, -0.764057, 1.570796, 1.701646],accel_mss,speed_ms,0,blend_radius_m)
    movel([0.130636, -1.372371, -2.575899, -0.764118, 1.570796, 1.701432],accel_mss,speed_ms,0,blend_radius_m)
    movel([0.130393, -1.372200, -2.576018, -0.764171, 1.570796, 1.701189],accel_mss,speed_ms,0,blend_radius_m)
    movel([0.130119, -1.372060, -2.576115, -0.764213, 1.570796, 1.700915],accel_mss,speed_ms,0,blend_radius_m)
    movel([0.129822, -1.371956, -2.576187, -0.764245, 1.570796, 1.700619],accel_mss,speed_ms,0,blend_radius_m)
    movel([0.129504, -1.371884, -2.576238, -0.764267, 1.570796, 1.700301],accel_mss,speed_ms,0,blend_radius_m)
    movel([0.129145, -1.371843, -2.576266, -0.764280, 1.570796, 1.699941],accel_mss,speed_ms,0,blend_radius_m)
    movel([0.128766, -1.371835, -2.576272, -0.764282, 1.570796, 1.699563],accel_mss,speed_ms,0,blend_radius_m)
    movel([0.128371, -1.371859, -2.576255, -0.764275, 1.570796, 1.699167],accel_mss,speed_ms,0,blend_radius_m)
    movel([0.127963, -1.371916, -2.576216, -0.764258, 1.570796, 1.698759],accel_mss,speed_ms,0,blend_radius_m)
    movel([0.127548, -1.372007, -2.576152, -0.764230, 1.570796, 1.698344],accel_mss,speed_ms,0,blend_radius_m)
    movel([0.127128, -1.372129, -2.576068, -0.764192, 1.570796, 1.697925],accel_mss,speed_ms,0,blend_radius_m)
    movel([0.126704, -1.372282, -2.575961, -0.764145, 1.570796, 1.697501],accel_mss,speed_ms,0,blend_radius_m)
    movel([0.126281, -1.372467, -2.575833, -0.764089, 1.570796, 1.697077],accel_mss,speed_ms,0,blend_radius_m)
    movel([0.125863, -1.372678, -2.575686, -0.764024, 1.570796, 1.696659],accel_mss,speed_ms,0,blend_radius_m)
    movel([0.125451, -1.372920, -2.575518, -0.763951, 1.570796, 1.696247],accel_mss,speed_ms,0,blend_radius_m)
    movel([0.125052, -1.373184, -2.575335, -0.763871, 1.570796, 1.695849],accel_mss,speed_ms,0,blend_radius_m)
    movel([0.124668, -1.373469, -2.575136, -0.763784, 1.570796, 1.695464],accel_mss,speed_ms,0,blend_radius_m)
    movel([0.124306, -1.373772, -2.574926, -0.763692, 1.570796, 1.695102],accel_mss,speed_ms,0,blend_radius_m)
    movel([0.123976, -1.374083, -2.574709, -0.763597, 1.570796, 1.694773],accel_mss,speed_ms,0,blend_radius_m)
    movel([0.123669, -1.374411, -2.574480, -0.763498, 1.570796, 1.694465],accel_mss,speed_ms,0,blend_radius_m)
    movel([0.123388, -1.374752, -2.574242, -0.763395, 1.570796, 1.694185],accel_mss,speed_ms,0,blend_radius_m)
    movel([0.123138, -1.375103, -2.573997, -0.763289, 1.570796, 1.693935],accel_mss,speed_ms,0,blend_radius_m)
    movel([0.122919, -1.375461, -2.573747, -0.763181, 1.570796, 1.693715],accel_mss,speed_ms,0,blend_radius_m)
    movel([0.122730, -1.375825, -2.573492, -0.763072, 1.570796, 1.693526],accel_mss,speed_ms,0,blend_radius_m)
    movel([0.122584, -1.376176, -2.573246, -0.762966, 1.570796, 1.693380],accel_mss,speed_ms,0,blend_radius_m)
    movel([0.122474, -1.376528, -2.573000, -0.762861, 1.570796, 1.693270],accel_mss,speed_ms,0,blend_radius_m)
    movel([0.122404, -1.376869, -2.572761, -0.762759, 1.570796, 1.693201],accel_mss,speed_ms,0,blend_radius_m)
    movel([0.122379, -1.377184, -2.572541, -0.762665, 1.570796, 1.693176],accel_mss,speed_ms,0,blend_radius_m)
    movel([0.122395, -1.377483, -2.572330, -0.762575, 1.570796, 1.693191],accel_mss,speed_ms,0,blend_radius_m)
    movel([0.122450, -1.377779, -2.572123, -0.762487, 1.570796, 1.693246],accel_mss,speed_ms,0,blend_radius_m)
    movel([0.122546, -1.378055, -2.571929, -0.762405, 1.570796, 1.693342],accel_mss,speed_ms,0,blend_radius_m)
    movel([0.122696, -1.378336, -2.571732, -0.762322, 1.570796, 1.693493],accel_mss,speed_ms,0,blend_radius_m)
    movel([0.122919, -1.378633, -2.571523, -0.762233, 1.570796, 1.693715],accel_mss,speed_ms,0,blend_radius_m)
    movel([0.123176, -1.378894, -2.571339, -0.762156, 1.570796, 1.693972],accel_mss,speed_ms,0,blend_radius_m)
    movel([0.123446, -1.379106, -2.571190, -0.762093, 1.570796, 1.694242],accel_mss,speed_ms,0,blend_radius_m)
    movel([0.123746, -1.379276, -2.571070, -0.762043, 1.570796, 1.694543],accel_mss,speed_ms,0,blend_radius_m)
    movel([0.124073, -1.379409, -2.570976, -0.762004, 1.570796, 1.694870],accel_mss,speed_ms,0,blend_radius_m)
    movel([0.124432, -1.379505, -2.570908, -0.761975, 1.570796, 1.695228],accel_mss,speed_ms,0,blend_radius_m)
    movel([0.124813, -1.379564, -2.570867, -0.761958, 1.570796, 1.695609],accel_mss,speed_ms,0,blend_radius_m)
    movel([0.125218, -1.379583, -2.570853, -0.761952, 1.570796, 1.696015],accel_mss,speed_ms,0,blend_radius_m)
    movel([0.125639, -1.379561, -2.570869, -0.761959, 1.570796, 1.696436],accel_mss,speed_ms,0,blend_radius_m)
    movel([0.126071, -1.379500, -2.570912, -0.761977, 1.570796, 1.696867],accel_mss,speed_ms,0,blend_radius_m)
    movel([0.126513, -1.379398, -2.570984, -0.762007, 1.570796, 1.697309],accel_mss,speed_ms,0,blend_radius_m)
    movel([0.126958, -1.379258, -2.571082, -0.762048, 1.570796, 1.697754],accel_mss,speed_ms,0,blend_radius_m)
    movel([0.127409, -1.379081, -2.571207, -0.762100, 1.570796, 1.698205],accel_mss,speed_ms,0,blend_radius_m)
    movel([0.127853, -1.378866, -2.571359, -0.762164, 1.570796, 1.698649],accel_mss,speed_ms,0,blend_radius_m)
    movel([0.128286, -1.378620, -2.571532, -0.762237, 1.570796, 1.699082],accel_mss,speed_ms,0,blend_radius_m)
    movel([0.128709, -1.378339, -2.571729, -0.762321, 1.570796, 1.699505],accel_mss,speed_ms,0,blend_radius_m)
    movel([0.129118, -1.378025, -2.571950, -0.762414, 1.570796, 1.699914],accel_mss,speed_ms,0,blend_radius_m)
    movel([0.129500, -1.377687, -2.572187, -0.762514, 1.570796, 1.700296],accel_mss,speed_ms,0,blend_radius_m)
    movel([0.129856, -1.377328, -2.572439, -0.762621, 1.570796, 1.700652],accel_mss,speed_ms,0,blend_radius_m)
    movel([0.130182, -1.376949, -2.572705, -0.762735, 1.570796, 1.700978],accel_mss,speed_ms,0,blend_radius_m)
    movel([0.130476, -1.376553, -2.572983, -0.762853, 1.570796, 1.701273],accel_mss,speed_ms,0,blend_radius_m)
    movel([0.130732, -1.376147, -2.573267, -0.762975, 1.570796, 1.701528],accel_mss,speed_ms,0,blend_radius_m)
    movel([0.130948, -1.375737, -2.573554, -0.763098, 1.570796, 1.701744],accel_mss,speed_ms,0,blend_radius_m)
    movel([0.131115, -1.375345, -2.573828, -0.763216, 1.570796, 1.701911],accel_mss,speed_ms,0,blend_radius_m)
    movel([0.131241, -1.374953, -2.574102, -0.763334, 1.570796, 1.702037],accel_mss,speed_ms,0,blend_radius_m)
    movel([0.131327, -1.374556, -2.574379, -0.763454, 1.570796, 1.702124],accel_mss,speed_ms,0,blend_radius_m)
    movel([0.131361, -1.374218, -2.574614, -0.763556, 1.570796, 1.702157],accel_mss,speed_ms,0,blend_radius_m)
    movel([0.131341, -1.373821, -2.574891, -0.763677, 1.570796, 1.702138],accel_mss,speed_ms,0,blend_radius_m)
    movel([0.131273, -1.373422, -2.575169, -0.763798, 1.570796, 1.702069],accel_mss,speed_ms,0,blend_radius_m)
    movel([0.131164, -1.373070, -2.575414, -0.763905, 1.570796, 1.701961],accel_mss,speed_ms,0,blend_radius_m)
    movel([0.131028, -1.372804, -2.575599, -0.763986, 1.570796, 1.701824],accel_mss,speed_ms,0,blend_radius_m)
    movel([0.131028, -1.375603, -2.576869, -0.759917, 1.570796, 1.701824],accel_mss,speed_ms,0,blend_radius_m)
    movel([0.130850, -1.375374, -2.577029, -0.759986, 1.570796, 1.701646],accel_mss,speed_ms,0,blend_radius_m)
    movel([0.130636, -1.375172, -2.577170, -0.760047, 1.570796, 1.701432],accel_mss,speed_ms,0,blend_radius_m)
    movel([0.130393, -1.375001, -2.577289, -0.760099, 1.570796, 1.701189],accel_mss,speed_ms,0,blend_radius_m)
    movel([0.130119, -1.374862, -2.577386, -0.760141, 1.570796, 1.700915],accel_mss,speed_ms,0,blend_radius_m)
    movel([0.129822, -1.374758, -2.577458, -0.760173, 1.570796, 1.700619],accel_mss,speed_ms,0,blend_radius_m)
    movel([0.129504, -1.374685, -2.577509, -0.760195, 1.570796, 1.700301],accel_mss,speed_ms,0,blend_radius_m)
    movel([0.129145, -1.374645, -2.577537, -0.760207, 1.570796, 1.699941],accel_mss,speed_ms,0,blend_radius_m)
    movel([0.128766, -1.374637, -2.577543, -0.760209, 1.570796, 1.699563],accel_mss,speed_ms,0,blend_radius_m)
    movel([0.128371, -1.374661, -2.577526, -0.760202, 1.570796, 1.699167],accel_mss,speed_ms,0,blend_radius_m)
    movel([0.127963, -1.374718, -2.577486, -0.760185, 1.570796, 1.698759],accel_mss,speed_ms,0,blend_radius_m)
    movel([0.127548, -1.374809, -2.577423, -0.760157, 1.570796, 1.698344],accel_mss,speed_ms,0,blend_radius_m)
    movel([0.127128, -1.374930, -2.577338, -0.760120, 1.570796, 1.697925],accel_mss,speed_ms,0,blend_radius_m)
    movel([0.126704, -1.375083, -2.577232, -0.760074, 1.570796, 1.697501],accel_mss,speed_ms,0,blend_radius_m)
    movel([0.126281, -1.375268, -2.577103, -0.760018, 1.570796, 1.697077],accel_mss,speed_ms,0,blend_radius_m)
    movel([0.125863, -1.375478, -2.576956, -0.759955, 1.570796, 1.696659],accel_mss,speed_ms,0,blend_radius_m)
    movel([0.125451, -1.375720, -2.576788, -0.759882, 1.570796, 1.696247],accel_mss,speed_ms,0,blend_radius_m)
    movel([0.125052, -1.375982, -2.576604, -0.759803, 1.570796, 1.695849],accel_mss,speed_ms,0,blend_radius_m)
    movel([0.124668, -1.376267, -2.576405, -0.759717, 1.570796, 1.695464],accel_mss,speed_ms,0,blend_radius_m)
    movel([0.124306, -1.376569, -2.576194, -0.759626, 1.570796, 1.695102],accel_mss,speed_ms,0,blend_radius_m)
    movel([0.123976, -1.376880, -2.575977, -0.759533, 1.570796, 1.694773],accel_mss,speed_ms,0,blend_radius_m)
    movel([0.123669, -1.377207, -2.575747, -0.759434, 1.570796, 1.694465],accel_mss,speed_ms,0,blend_radius_m)
    movel([0.123388, -1.377547, -2.575509, -0.759333, 1.570796, 1.694185],accel_mss,speed_ms,0,blend_radius_m)
    movel([0.123138, -1.377898, -2.575263, -0.759228, 1.570796, 1.693935],accel_mss,speed_ms,0,blend_radius_m)
    movel([0.122919, -1.378255, -2.575013, -0.759122, 1.570796, 1.693715],accel_mss,speed_ms,0,blend_radius_m)
    movel([0.122730, -1.378618, -2.574757, -0.759013, 1.570796, 1.693526],accel_mss,speed_ms,0,blend_radius_m)
    movel([0.122584, -1.378969, -2.574511, -0.758909, 1.570796, 1.693380],accel_mss,speed_ms,0,blend_radius_m)
    movel([0.122474, -1.379320, -2.574264, -0.758805, 1.570796, 1.693270],accel_mss,speed_ms,0,blend_radius_m)
    movel([0.122404, -1.379660, -2.574025, -0.758704, 1.570796, 1.693201],accel_mss,speed_ms,0,blend_radius_m)
    movel([0.122379, -1.379974, -2.573804, -0.758611, 1.570796, 1.693176],accel_mss,speed_ms,0,blend_radius_m)
    movel([0.122395, -1.380273, -2.573594, -0.758523, 1.570796, 1.693191],accel_mss,speed_ms,0,blend_radius_m)
    movel([0.122450, -1.380567, -2.573386, -0.758436, 1.570796, 1.693246],accel_mss,speed_ms,0,blend_radius_m)
    movel([0.122546, -1.380843, -2.573191, -0.758355, 1.570796, 1.693342],accel_mss,speed_ms,0,blend_radius_m)
    movel([0.122696, -1.381123, -2.572994, -0.758272, 1.570796, 1.693493],accel_mss,speed_ms,0,blend_radius_m)
    movel([0.122919, -1.381420, -2.572784, -0.758185, 1.570796, 1.693715],accel_mss,speed_ms,0,blend_radius_m)
    movel([0.123176, -1.381680, -2.572600, -0.758109, 1.570796, 1.693972],accel_mss,speed_ms,0,blend_radius_m)
    movel([0.123446, -1.381891, -2.572451, -0.758047, 1.570796, 1.694242],accel_mss,speed_ms,0,blend_radius_m)
    movel([0.123746, -1.382061, -2.572331, -0.757997, 1.570796, 1.694543],accel_mss,speed_ms,0,blend_radius_m)
    movel([0.124073, -1.382194, -2.572237, -0.757958, 1.570796, 1.694870],accel_mss,speed_ms,0,blend_radius_m)
    movel([0.124432, -1.382290, -2.572169, -0.757930, 1.570796, 1.695228],accel_mss,speed_ms,0,blend_radius_m)
    movel([0.124813, -1.382349, -2.572127, -0.757913, 1.570796, 1.695609],accel_mss,speed_ms,0,blend_radius_m)
    movel([0.125218, -1.382368, -2.572114, -0.757908, 1.570796, 1.696015],accel_mss,speed_ms,0,blend_radius_m)
    movel([0.125639, -1.382345, -2.572130, -0.757914, 1.570796, 1.696436],accel_mss,speed_ms,0,blend_radius_m)
    movel([0.126071, -1.382284, -2.572173, -0.757932, 1.570796, 1.696867],accel_mss,speed_ms,0,blend_radius_m)
    movel([0.126513, -1.382183, -2.572244, -0.757962, 1.570796, 1.697309],accel_mss,speed_ms,0,blend_radius_m)
    movel([0.126958, -1.382044, -2.572343, -0.758002, 1.570796, 1.697754],accel_mss,speed_ms,0,blend_radius_m)
    movel([0.127409, -1.381867, -2.572468, -0.758054, 1.570796, 1.698205],accel_mss,speed_ms,0,blend_radius_m)
    movel([0.127853, -1.381652, -2.572620, -0.758117, 1.570796, 1.698649],accel_mss,speed_ms,0,blend_radius_m)
    movel([0.128286, -1.381407, -2.572793, -0.758189, 1.570796, 1.699082],accel_mss,speed_ms,0,blend_radius_m)
    movel([0.128709, -1.381126, -2.572991, -0.758271, 1.570796, 1.699505],accel_mss,speed_ms,0,blend_radius_m)
    movel([0.129118, -1.380813, -2.573212, -0.758363, 1.570796, 1.699914],accel_mss,speed_ms,0,blend_radius_m)
    movel([0.129500, -1.380476, -2.573450, -0.758463, 1.570796, 1.700296],accel_mss,speed_ms,0,blend_radius_m)
    movel([0.129856, -1.380118, -2.573703, -0.758569, 1.570796, 1.700652],accel_mss,speed_ms,0,blend_radius_m)
    movel([0.130182, -1.379740, -2.573969, -0.758680, 1.570796, 1.700978],accel_mss,speed_ms,0,blend_radius_m)
    movel([0.130476, -1.379344, -2.574247, -0.758798, 1.570796, 1.701273],accel_mss,speed_ms,0,blend_radius_m)
    movel([0.130732, -1.378939, -2.574532, -0.758918, 1.570796, 1.701528],accel_mss,speed_ms,0,blend_radius_m)
    movel([0.130948, -1.378530, -2.574820, -0.759040, 1.570796, 1.701744],accel_mss,speed_ms,0,blend_radius_m)
    movel([0.131115, -1.378139, -2.575094, -0.759156, 1.570796, 1.701911],accel_mss,speed_ms,0,blend_radius_m)
    movel([0.131241, -1.377748, -2.575369, -0.759273, 1.570796, 1.702037],accel_mss,speed_ms,0,blend_radius_m)
    movel([0.131327, -1.377351, -2.575646, -0.759391, 1.570796, 1.702124],accel_mss,speed_ms,0,blend_radius_m)
    movel([0.131361, -1.377015, -2.575882, -0.759492, 1.570796, 1.702157],accel_mss,speed_ms,0,blend_radius_m)
    movel([0.131341, -1.376618, -2.576160, -0.759611, 1.570796, 1.702138],accel_mss,speed_ms,0,blend_radius_m)
    movel([0.131273, -1.376221, -2.576438, -0.759731, 1.570796, 1.702069],accel_mss,speed_ms,0,blend_radius_m)
    movel([0.131164, -1.375869, -2.576683, -0.759837, 1.570796, 1.701961],accel_mss,speed_ms,0,blend_radius_m)
    movel([0.131028, -1.375603, -2.576869, -0.759917, 1.570796, 1.701824],accel_mss,speed_ms,0,blend_radius_m)
    movel([0.131028, -1.343086, -2.561242, -0.808061, 1.570796, 1.701824],accel_mss,speed_ms,0,blend_radius_m)
    speed_ms = 1.000
    movel([0.135704, -1.338118, -2.564530, -0.809741, 1.570796, 1.706501],accel_mss,speed_ms,0,blend_radius_m)
    speed_ms = 0.008
    movel([0.135704, -1.364599, -2.577427, -0.770363, 1.570796, 1.706501],accel_mss,speed_ms,0,blend_radius_m)
    speed_ms = 0.003
    movel([0.135704, -1.367941, -2.578962, -0.765485, 1.570796, 1.706501],accel_mss,speed_ms,0,blend_radius_m)
    speed_ms = 0.008
    movel([0.132243, -1.368831, -2.578349, -0.765209, 1.570796, 1.703039],accel_mss,speed_ms,0,blend_radius_m)
    movel([0.133489, -1.372007, -2.576153, -0.764230, 1.570796, 1.704286],accel_mss,speed_ms,0,blend_radius_m)
    movel([0.133900, -1.372999, -2.575463, -0.763927, 1.570796, 1.704697],accel_mss,speed_ms,0,blend_radius_m)
    movel([0.134187, -1.373631, -2.575024, -0.763735, 1.570796, 1.704983],accel_mss,speed_ms,0,blend_radius_m)
    movel([0.134528, -1.374312, -2.574549, -0.763528, 1.570796, 1.705325],accel_mss,speed_ms,0,blend_radius_m)
    movel([0.134698, -1.374634, -2.574324, -0.763431, 1.570796, 1.705494],accel_mss,speed_ms,0,blend_radius_m)
    movel([0.134972, -1.374403, -2.574485, -0.763500, 1.570796, 1.705768],accel_mss,speed_ms,0,blend_radius_m)
    movel([0.135456, -1.373576, -2.575061, -0.763751, 1.570796, 1.706253],accel_mss,speed_ms,0,blend_radius_m)
    movel([0.136749, -1.371331, -2.576621, -0.764437, 1.570796, 1.707545],accel_mss,speed_ms,0,blend_radius_m)
    movel([0.139168, -1.367060, -2.579568, -0.765761, 1.570796, 1.709964],accel_mss,speed_ms,0,blend_radius_m)
    movel([0.135704, -1.367941, -2.578962, -0.765485, 1.570796, 1.706501],accel_mss,speed_ms,0,blend_radius_m)
    movel([0.135704, -1.370752, -2.580239, -0.761398, 1.570796, 1.706501],accel_mss,speed_ms,0,blend_radius_m)
    movel([0.132243, -1.371640, -2.579625, -0.761125, 1.570796, 1.703039],accel_mss,speed_ms,0,blend_radius_m)
    movel([0.133489, -1.374808, -2.577423, -0.760157, 1.570796, 1.704286],accel_mss,speed_ms,0,blend_radius_m)
    movel([0.133900, -1.375798, -2.576733, -0.759858, 1.570796, 1.704697],accel_mss,speed_ms,0,blend_radius_m)
    movel([0.134187, -1.376429, -2.576292, -0.759668, 1.570796, 1.704983],accel_mss,speed_ms,0,blend_radius_m)
    movel([0.134528, -1.377109, -2.575816, -0.759464, 1.570796, 1.705325],accel_mss,speed_ms,0,blend_radius_m)
    movel([0.134698, -1.377430, -2.575591, -0.759368, 1.570796, 1.705494],accel_mss,speed_ms,0,blend_radius_m)
    movel([0.134972, -1.377200, -2.575753, -0.759437, 1.570796, 1.705768],accel_mss,speed_ms,0,blend_radius_m)
    movel([0.135456, -1.376374, -2.576330, -0.759685, 1.570796, 1.706253],accel_mss,speed_ms,0,blend_radius_m)
    movel([0.136749, -1.374134, -2.577893, -0.760362, 1.570796, 1.707545],accel_mss,speed_ms,0,blend_radius_m)
    movel([0.139168, -1.369873, -2.580846, -0.761670, 1.570796, 1.709964],accel_mss,speed_ms,0,blend_radius_m)
    movel([0.135704, -1.370752, -2.580239, -0.761398, 1.570796, 1.706501],accel_mss,speed_ms,0,blend_radius_m)
    movel([0.135704, -1.338118, -2.564530, -0.809741, 1.570796, 1.706501],accel_mss,speed_ms,0,blend_radius_m)
    speed_ms = 1.000
    movel([0.112823, -1.351262, -2.555758, -0.805368, 1.570796, 1.683619],accel_mss,speed_ms,0,blend_radius_m)
    speed_ms = 0.008
    movel([0.112823, -1.377494, -2.568480, -0.766416, 1.570796, 1.683619],accel_mss,speed_ms,0,blend_radius_m)
    speed_ms = 0.003
    movel([0.112823, -1.380802, -2.569994, -0.761594, 1.570796, 1.683619],accel_mss,speed_ms,0,blend_radius_m)
    speed_ms = 0.008
    movel([0.111626, -1.381124, -2.569766, -0.761499, 1.570796, 1.682422],accel_mss,speed_ms,0,blend_radius_m)
    movel([0.112710, -1.372739, -2.575644, -0.764006, 1.570796, 1.683506],accel_mss,speed_ms,0,blend_radius_m)
    movel([0.115128, -1.372082, -2.576100, -0.764207, 1.570796, 1.685924],accel_mss,speed_ms,0,blend_radius_m)
    movel([0.114020, -1.380481, -2.570221, -0.761688, 1.570796, 1.684816],accel_mss,speed_ms,0,blend_radius_m)
    movel([0.112823, -1.380802, -2.569994, -0.761594, 1.570796, 1.683619],accel_mss,speed_ms,0,blend_radius_m)
    movel([0.112823, -1.383583, -2.571252, -0.757554, 1.570796, 1.683619],accel_mss,speed_ms,0,blend_radius_m)
    movel([0.111626, -1.383905, -2.571024, -0.757460, 1.570796, 1.682422],accel_mss,speed_ms,0,blend_radius_m)
    movel([0.112710, -1.375539, -2.576913, -0.759936, 1.570796, 1.683506],accel_mss,speed_ms,0,blend_radius_m)
    movel([0.115128, -1.374883, -2.577371, -0.760135, 1.570796, 1.685924],accel_mss,speed_ms,0,blend_radius_m)
    movel([0.114020, -1.383263, -2.571479, -0.757647, 1.570796, 1.684816],accel_mss,speed_ms,0,blend_radius_m)
    movel([0.112823, -1.383583, -2.571252, -0.757554, 1.570796, 1.683619],accel_mss,speed_ms,0,blend_radius_m)
    movel([0.112823, -1.351262, -2.555758, -0.805368, 1.570796, 1.683619],accel_mss,speed_ms,0,blend_radius_m)
    speed_ms = 1.000
    movel([0.180901, -1.303040, -2.586825, -0.822524, 1.570796, 1.751698],accel_mss,speed_ms,0,blend_radius_m)
    speed_ms = 0.008
    movel([0.180901, -1.330151, -2.600194, -0.782044, 1.570796, 1.751698],accel_mss,speed_ms,0,blend_radius_m)
    speed_ms = 0.003
    movel([0.180901, -1.333580, -2.601787, -0.777022, 1.570796, 1.751698],accel_mss,speed_ms,0,blend_radius_m)
    speed_ms = 0.008
    movel([0.180599, -1.333907, -2.601578, -0.776904, 1.570796, 1.751396],accel_mss,speed_ms,0,blend_radius_m)
    movel([0.180282, -1.334226, -2.601373, -0.776790, 1.570796, 1.751078],accel_mss,speed_ms,0,blend_radius_m)
    movel([0.179952, -1.334532, -2.601177, -0.776680, 1.570796, 1.750748],accel_mss,speed_ms,0,blend_radius_m)
    movel([0.179609, -1.334824, -2.600989, -0.776576, 1.570796, 1.750406],accel_mss,speed_ms,0,blend_radius_m)
    movel([0.179219, -1.335135, -2.600789, -0.776464, 1.570796, 1.750015],accel_mss,speed_ms,0,blend_radius_m)
    movel([0.178734, -1.335498, -2.600556, -0.776335, 1.570796, 1.749531],accel_mss,speed_ms,0,blend_radius_m)
    movel([0.178263, -1.335832, -2.600341, -0.776216, 1.570796, 1.749059],accel_mss,speed_ms,0,blend_radius_m)
    movel([0.177786, -1.336156, -2.600132, -0.776100, 1.570796, 1.748582],accel_mss,speed_ms,0,blend_radius_m)
    movel([0.177305, -1.336466, -2.599933, -0.775990, 1.570796, 1.748101],accel_mss,speed_ms,0,blend_radius_m)
    movel([0.176780, -1.336783, -2.599728, -0.775877, 1.570796, 1.747576],accel_mss,speed_ms,0,blend_radius_m)
    movel([0.176259, -1.337087, -2.599532, -0.775770, 1.570796, 1.747055],accel_mss,speed_ms,0,blend_radius_m)
    movel([0.175730, -1.337376, -2.599345, -0.775667, 1.570796, 1.746526],accel_mss,speed_ms,0,blend_radius_m)
    movel([0.175208, -1.337649, -2.599170, -0.775571, 1.570796, 1.746004],accel_mss,speed_ms,0,blend_radius_m)
    movel([0.174677, -1.337912, -2.598999, -0.775478, 1.570796, 1.745474],accel_mss,speed_ms,0,blend_radius_m)
    movel([0.174137, -1.338164, -2.598836, -0.775389, 1.570796, 1.744933],accel_mss,speed_ms,0,blend_radius_m)
    movel([0.173589, -1.338404, -2.598681, -0.775304, 1.570796, 1.744385],accel_mss,speed_ms,0,blend_radius_m)
    movel([0.172982, -1.338654, -2.598519, -0.775216, 1.570796, 1.743779],accel_mss,speed_ms,0,blend_radius_m)
    movel([0.172372, -1.338888, -2.598368, -0.775133, 1.570796, 1.743168],accel_mss,speed_ms,0,blend_radius_m)
    movel([0.171706, -1.339126, -2.598214, -0.775050, 1.570796, 1.742502],accel_mss,speed_ms,0,blend_radius_m)
    movel([0.171044, -1.339343, -2.598073, -0.774973, 1.570796, 1.741841],accel_mss,speed_ms,0,blend_radius_m)
    movel([0.170397, -1.339538, -2.597946, -0.774905, 1.570796, 1.741193],accel_mss,speed_ms,0,blend_radius_m)
    movel([0.169698, -1.339734, -2.597819, -0.774836, 1.570796, 1.740494],accel_mss,speed_ms,0,blend_radius_m)
    movel([0.169002, -1.339910, -2.597705, -0.774774, 1.570796, 1.739798],accel_mss,speed_ms,0,blend_radius_m)
    movel([0.168306, -1.340074, -2.597598, -0.774717, 1.570796, 1.739103],accel_mss,speed_ms,0,blend_radius_m)
    movel([0.167053, -1.340329, -2.597433, -0.774627, 1.570796, 1.737850],accel_mss,speed_ms,0,blend_radius_m)
    movel([0.166310, -1.340458, -2.597349, -0.774582, 1.570796, 1.737106],accel_mss,speed_ms,0,blend_radius_m)
    movel([0.166015, -1.340496, -2.597324, -0.774569, 1.570796, 1.736811],accel_mss,speed_ms,0,blend_radius_m)
    movel([0.165607, -1.340424, -2.597371, -0.774594, 1.570796, 1.736403],accel_mss,speed_ms,0,blend_radius_m)
    movel([0.165439, -1.340275, -2.597468, -0.774646, 1.570796, 1.736235],accel_mss,speed_ms,0,blend_radius_m)
    movel([0.165520, -1.339246, -2.598136, -0.775007, 1.570796, 1.736316],accel_mss,speed_ms,0,blend_radius_m)
    movel([0.165676, -1.338271, -2.598767, -0.775351, 1.570796, 1.736472],accel_mss,speed_ms,0,blend_radius_m)
    movel([0.165834, -1.337469, -2.599286, -0.775634, 1.570796, 1.736631],accel_mss,speed_ms,0,blend_radius_m)
    movel([0.166469, -1.334534, -2.601176, -0.776680, 1.570796, 1.737266],accel_mss,speed_ms,0,blend_radius_m)
    movel([0.181058, -1.329600, -2.604326, -0.778463, 1.570796, 1.751855],accel_mss,speed_ms,0,blend_radius_m)
    movel([0.181396, -1.329497, -2.604392, -0.778500, 1.570796, 1.752193],accel_mss,speed_ms,0,blend_radius_m)
    movel([0.181732, -1.329409, -2.604448, -0.778532, 1.570796, 1.752528],accel_mss,speed_ms,0,blend_radius_m)
    movel([0.182074, -1.329337, -2.604493, -0.778559, 1.570796, 1.752870],accel_mss,speed_ms,0,blend_radius_m)
    movel([0.182360, -1.329293, -2.604522, -0.778575, 1.570796, 1.753157],accel_mss,speed_ms,0,blend_radius_m)
    movel([0.182621, -1.329361, -2.604478, -0.778550, 1.570796, 1.753418],accel_mss,speed_ms,0,blend_radius_m)
    movel([0.182727, -1.329582, -2.604338, -0.778469, 1.570796, 1.753523],accel_mss,speed_ms,0,blend_radius_m)
    movel([0.182725, -1.329911, -2.604129, -0.778349, 1.570796, 1.753521],accel_mss,speed_ms,0,blend_radius_m)
    movel([0.182683, -1.330255, -2.603910, -0.778224, 1.570796, 1.753479],accel_mss,speed_ms,0,blend_radius_m)
    movel([0.182610, -1.330577, -2.603705, -0.778107, 1.570796, 1.753406],accel_mss,speed_ms,0,blend_radius_m)
    movel([0.182464, -1.331039, -2.603411, -0.777939, 1.570796, 1.753260],accel_mss,speed_ms,0,blend_radius_m)
    movel([0.182322, -1.331431, -2.603161, -0.777797, 1.570796, 1.753118],accel_mss,speed_ms,0,blend_radius_m)
    movel([0.182204, -1.331708, -2.602984, -0.777697, 1.570796, 1.753000],accel_mss,speed_ms,0,blend_radius_m)
    movel([0.182056, -1.332009, -2.602792, -0.777588, 1.570796, 1.752852],accel_mss,speed_ms,0,blend_radius_m)
    movel([0.181886, -1.332305, -2.602603, -0.777481, 1.570796, 1.752682],accel_mss,speed_ms,0,blend_radius_m)
    movel([0.181703, -1.332584, -2.602425, -0.777380, 1.570796, 1.752499],accel_mss,speed_ms,0,blend_radius_m)
    movel([0.181500, -1.332860, -2.602248, -0.777281, 1.570796, 1.752296],accel_mss,speed_ms,0,blend_radius_m)
    movel([0.181207, -1.333223, -2.602016, -0.777150, 1.570796, 1.752004],accel_mss,speed_ms,0,blend_radius_m)
    movel([0.180901, -1.333580, -2.601787, -0.777022, 1.570796, 1.751698],accel_mss,speed_ms,0,blend_radius_m)
    movel([0.180901, -1.336465, -2.603112, -0.772812, 1.570796, 1.751698],accel_mss,speed_ms,0,blend_radius_m)
    movel([0.180599, -1.336791, -2.602902, -0.772696, 1.570796, 1.751396],accel_mss,speed_ms,0,blend_radius_m)
    movel([0.180282, -1.337109, -2.602697, -0.772582, 1.570796, 1.751078],accel_mss,speed_ms,0,blend_radius_m)
    movel([0.179952, -1.337415, -2.602501, -0.772474, 1.570796, 1.750748],accel_mss,speed_ms,0,blend_radius_m)
    movel([0.179609, -1.337707, -2.602312, -0.772370, 1.570796, 1.750406],accel_mss,speed_ms,0,blend_radius_m)
    movel([0.179219, -1.338017, -2.602112, -0.772260, 1.570796, 1.750015],accel_mss,speed_ms,0,blend_radius_m)
    movel([0.178734, -1.338379, -2.601878, -0.772132, 1.570796, 1.749531],accel_mss,speed_ms,0,blend_radius_m)
    movel([0.178263, -1.338712, -2.601663, -0.772014, 1.570796, 1.749059],accel_mss,speed_ms,0,blend_radius_m)
    movel([0.177786, -1.339036, -2.601453, -0.771900, 1.570796, 1.748582],accel_mss,speed_ms,0,blend_radius_m)
    movel([0.177305, -1.339345, -2.601254, -0.771791, 1.570796, 1.748101],accel_mss,speed_ms,0,blend_radius_m)
    movel([0.176780, -1.339662, -2.601048, -0.771679, 1.570796, 1.747576],accel_mss,speed_ms,0,blend_radius_m)
    movel([0.176259, -1.339965, -2.600852, -0.771572, 1.570796, 1.747055],accel_mss,speed_ms,0,blend_radius_m)
    movel([0.175730, -1.340254, -2.600665, -0.771471, 1.570796, 1.746526],accel_mss,speed_ms,0,blend_radius_m)
    movel([0.175208, -1.340525, -2.600489, -0.771375, 1.570796, 1.746004],accel_mss,speed_ms,0,blend_radius_m)
    movel([0.174677, -1.340788, -2.600318, -0.771283, 1.570796, 1.745474],accel_mss,speed_ms,0,blend_radius_m)
    movel([0.174137, -1.341039, -2.600155, -0.771195, 1.570796, 1.744933],accel_mss,speed_ms,0,blend_radius_m)
    movel([0.173589, -1.341279, -2.599999, -0.771111, 1.570796, 1.744385],accel_mss,speed_ms,0,blend_radius_m)
    movel([0.172982, -1.341529, -2.599837, -0.771024, 1.570796, 1.743779],accel_mss,speed_ms,0,blend_radius_m)
    movel([0.172372, -1.341762, -2.599685, -0.770942, 1.570796, 1.743168],accel_mss,speed_ms,0,blend_radius_m)
    movel([0.171706, -1.341999, -2.599531, -0.770859, 1.570796, 1.742502],accel_mss,speed_ms,0,blend_radius_m)
    movel([0.171044, -1.342216, -2.599390, -0.770784, 1.570796, 1.741841],accel_mss,speed_ms,0,blend_radius_m)
    movel([0.170397, -1.342411, -2.599262, -0.770716, 1.570796, 1.741193],accel_mss,speed_ms,0,blend_radius_m)
    movel([0.169698, -1.342606, -2.599135, -0.770648, 1.570796, 1.740494],accel_mss,speed_ms,0,blend_radius_m)
    movel([0.169002, -1.342782, -2.599020, -0.770586, 1.570796, 1.739798],accel_mss,speed_ms,0,blend_radius_m)
    movel([0.168306, -1.342946, -2.598914, -0.770530, 1.570796, 1.739103],accel_mss,speed_ms,0,blend_radius_m)
    movel([0.167053, -1.343200, -2.598748, -0.770441, 1.570796, 1.737850],accel_mss,speed_ms,0,blend_radius_m)
    movel([0.166310, -1.343329, -2.598664, -0.770396, 1.570796, 1.737106],accel_mss,speed_ms,0,blend_radius_m)
    movel([0.166015, -1.343367, -2.598639, -0.770383, 1.570796, 1.736811],accel_mss,speed_ms,0,blend_radius_m)
    movel([0.165607, -1.343295, -2.598686, -0.770408, 1.570796, 1.736403],accel_mss,speed_ms,0,blend_radius_m)
    movel([0.165439, -1.343146, -2.598783, -0.770460, 1.570796, 1.736235],accel_mss,speed_ms,0,blend_radius_m)
    movel([0.165520, -1.342119, -2.599453, -0.770817, 1.570796, 1.736316],accel_mss,speed_ms,0,blend_radius_m)
    movel([0.165676, -1.341146, -2.600085, -0.771158, 1.570796, 1.736472],accel_mss,speed_ms,0,blend_radius_m)
    movel([0.165834, -1.340346, -2.600605, -0.771438, 1.570796, 1.736631],accel_mss,speed_ms,0,blend_radius_m)
    movel([0.166469, -1.337417, -2.602499, -0.772473, 1.570796, 1.737266],accel_mss,speed_ms,0,blend_radius_m)
    movel([0.181058, -1.332493, -2.605657, -0.774239, 1.570796, 1.751855],accel_mss,speed_ms,0,blend_radius_m)
    movel([0.181396, -1.332391, -2.605722, -0.774276, 1.570796, 1.752193],accel_mss,speed_ms,0,blend_radius_m)
    movel([0.181732, -1.332303, -2.605778, -0.774308, 1.570796, 1.752528],accel_mss,speed_ms,0,blend_radius_m)
    movel([0.182074, -1.332231, -2.605824, -0.774334, 1.570796, 1.752870],accel_mss,speed_ms,0,blend_radius_m)
    movel([0.182360, -1.332186, -2.605852, -0.774350, 1.570796, 1.753157],accel_mss,speed_ms,0,blend_radius_m)
    movel([0.182621, -1.332255, -2.605809, -0.774325, 1.570796, 1.753418],accel_mss,speed_ms,0,blend_radius_m)
    movel([0.182727, -1.332476, -2.605668, -0.774245, 1.570796, 1.753523],accel_mss,speed_ms,0,blend_radius_m)
    movel([0.182725, -1.332803, -2.605459, -0.774127, 1.570796, 1.753521],accel_mss,speed_ms,0,blend_radius_m)
    movel([0.182683, -1.333147, -2.605239, -0.774003, 1.570796, 1.753479],accel_mss,speed_ms,0,blend_radius_m)
    movel([0.182610, -1.333468, -2.605034, -0.773887, 1.570796, 1.753406],accel_mss,speed_ms,0,blend_radius_m)
    movel([0.182464, -1.333929, -2.604739, -0.773721, 1.570796, 1.753260],accel_mss,speed_ms,0,blend_radius_m)
    movel([0.182322, -1.334320, -2.604489, -0.773580, 1.570796, 1.753118],accel_mss,speed_ms,0,blend_radius_m)
    movel([0.182204, -1.334597, -2.604311, -0.773480, 1.570796, 1.753000],accel_mss,speed_ms,0,blend_radius_m)
    movel([0.182056, -1.334897, -2.604119, -0.773373, 1.570796, 1.752852],accel_mss,speed_ms,0,blend_radius_m)
    movel([0.181886, -1.335193, -2.603930, -0.773267, 1.570796, 1.752682],accel_mss,speed_ms,0,blend_radius_m)
    movel([0.181703, -1.335471, -2.603751, -0.773167, 1.570796, 1.752499],accel_mss,speed_ms,0,blend_radius_m)
    movel([0.181500, -1.335747, -2.603574, -0.773068, 1.570796, 1.752296],accel_mss,speed_ms,0,blend_radius_m)
    movel([0.181207, -1.336109, -2.603341, -0.772939, 1.570796, 1.752004],accel_mss,speed_ms,0,blend_radius_m)
    movel([0.180901, -1.336465, -2.603112, -0.772812, 1.570796, 1.751698],accel_mss,speed_ms,0,blend_radius_m)
    movel([0.180901, -1.303040, -2.586825, -0.822524, 1.570796, 1.751698],accel_mss,speed_ms,0,blend_radius_m)
    speed_ms = 1.000
    movel([0.182539, -1.297981, -2.589909, -0.824499, 1.570796, 1.753336],accel_mss,speed_ms,0,blend_radius_m)
    speed_ms = 0.008
    movel([0.182539, -1.325178, -2.603347, -0.783864, 1.570796, 1.753336],accel_mss,speed_ms,0,blend_radius_m)
    speed_ms = 0.003
    movel([0.182539, -1.328619, -2.604949, -0.778821, 1.570796, 1.753336],accel_mss,speed_ms,0,blend_radius_m)
    speed_ms = 0.008
    movel([0.173197, -1.331762, -2.602950, -0.777677, 1.570796, 1.743994],accel_mss,speed_ms,0,blend_radius_m)
    movel([0.170898, -1.332531, -2.602458, -0.777399, 1.570796, 1.741694],accel_mss,speed_ms,0,blend_radius_m)
    movel([0.169571, -1.332964, -2.602182, -0.777243, 1.570796, 1.740368],accel_mss,speed_ms,0,blend_radius_m)
    movel([0.168187, -1.333373, -2.601920, -0.777096, 1.570796, 1.738984],accel_mss,speed_ms,0,blend_radius_m)
    movel([0.167669, -1.333514, -2.601830, -0.777045, 1.570796, 1.738465],accel_mss,speed_ms,0,blend_radius_m)
    movel([0.167277, -1.333604, -2.601772, -0.777013, 1.570796, 1.738074],accel_mss,speed_ms,0,blend_radius_m)
    movel([0.166905, -1.333673, -2.601728, -0.776988, 1.570796, 1.737701],accel_mss,speed_ms,0,blend_radius_m)
    movel([0.166564, -1.333718, -2.601699, -0.776972, 1.570796, 1.737360],accel_mss,speed_ms,0,blend_radius_m)
    movel([0.166485, -1.333521, -2.601825, -0.777043, 1.570796, 1.737282],accel_mss,speed_ms,0,blend_radius_m)
    movel([0.166795, -1.333293, -2.601971, -0.777125, 1.570796, 1.737592],accel_mss,speed_ms,0,blend_radius_m)
    movel([0.174123, -1.330792, -2.603568, -0.778029, 1.570796, 1.744919],accel_mss,speed_ms,0,blend_radius_m)
    movel([0.181377, -1.328362, -2.605112, -0.778915, 1.570796, 1.752174],accel_mss,speed_ms,0,blend_radius_m)
    movel([0.181869, -1.328221, -2.605201, -0.778967, 1.570796, 1.752665],accel_mss,speed_ms,0,blend_radius_m)
    movel([0.182357, -1.328098, -2.605279, -0.779012, 1.570796, 1.753153],accel_mss,speed_ms,0,blend_radius_m)
    movel([0.182620, -1.328096, -2.605280, -0.779013, 1.570796, 1.753417],accel_mss,speed_ms,0,blend_radius_m)
    movel([0.182827, -1.328261, -2.605175, -0.778952, 1.570796, 1.753623],accel_mss,speed_ms,0,blend_radius_m)
    movel([0.182639, -1.328573, -2.604978, -0.778838, 1.570796, 1.753435],accel_mss,speed_ms,0,blend_radius_m)
    movel([0.182539, -1.331514, -2.606281, -0.774594, 1.570796, 1.753336],accel_mss,speed_ms,0,blend_radius_m)
    movel([0.173197, -1.334651, -2.604277, -0.773461, 1.570796, 1.743994],accel_mss,speed_ms,0,blend_radius_m)
    movel([0.170898, -1.335419, -2.603785, -0.773186, 1.570796, 1.741694],accel_mss,speed_ms,0,blend_radius_m)
    movel([0.169571, -1.335850, -2.603508, -0.773031, 1.570796, 1.740368],accel_mss,speed_ms,0,blend_radius_m)
    movel([0.168187, -1.336258, -2.603245, -0.772886, 1.570796, 1.738984],accel_mss,speed_ms,0,blend_radius_m)
    movel([0.167669, -1.336399, -2.603154, -0.772835, 1.570796, 1.738465],accel_mss,speed_ms,0,blend_radius_m)
    movel([0.167277, -1.336489, -2.603097, -0.772803, 1.570796, 1.738074],accel_mss,speed_ms,0,blend_radius_m)
    movel([0.166905, -1.336558, -2.603053, -0.772779, 1.570796, 1.737701],accel_mss,speed_ms,0,blend_radius_m)
    movel([0.166564, -1.336603, -2.603023, -0.772763, 1.570796, 1.737360],accel_mss,speed_ms,0,blend_radius_m)
    movel([0.166485, -1.336406, -2.603150, -0.772833, 1.570796, 1.737282],accel_mss,speed_ms,0,blend_radius_m)
    movel([0.166795, -1.336179, -2.603296, -0.772914, 1.570796, 1.737592],accel_mss,speed_ms,0,blend_radius_m)
    movel([0.174123, -1.333683, -2.604897, -0.773809, 1.570796, 1.744919],accel_mss,speed_ms,0,blend_radius_m)
    movel([0.181377, -1.331258, -2.606444, -0.774687, 1.570796, 1.752174],accel_mss,speed_ms,0,blend_radius_m)
    movel([0.181869, -1.331117, -2.606534, -0.774739, 1.570796, 1.752665],accel_mss,speed_ms,0,blend_radius_m)
    movel([0.182357, -1.330995, -2.606611, -0.774783, 1.570796, 1.753153],accel_mss,speed_ms,0,blend_radius_m)
    movel([0.182620, -1.330992, -2.606613, -0.774784, 1.570796, 1.753417],accel_mss,speed_ms,0,blend_radius_m)
    movel([0.182827, -1.331158, -2.606508, -0.774724, 1.570796, 1.753623],accel_mss,speed_ms,0,blend_radius_m)
    movel([0.182639, -1.331468, -2.606310, -0.774611, 1.570796, 1.753435],accel_mss,speed_ms,0,blend_radius_m)
    movel([0.182539, -1.297981, -2.589909, -0.824499, 1.570796, 1.753336],accel_mss,speed_ms,0,blend_radius_m)
    speed_ms = 1.000
    movel([0.181339, -1.297216, -2.590373, -0.824800, 1.570796, 1.752135],accel_mss,speed_ms,0,blend_radius_m)
    speed_ms = 0.008
    movel([0.181339, -1.324426, -2.603821, -0.784142, 1.570796, 1.752135],accel_mss,speed_ms,0,blend_radius_m)
    speed_ms = 0.003
    movel([0.181339, -1.327869, -2.605424, -0.779096, 1.570796, 1.752135],accel_mss,speed_ms,0,blend_radius_m)
    speed_ms = 0.008
    movel([0.178454, -1.328846, -2.604805, -0.778738, 1.570796, 1.749250],accel_mss,speed_ms,0,blend_radius_m)
    movel([0.173139, -1.330638, -2.603666, -0.778085, 1.570796, 1.743935],accel_mss,speed_ms,0,blend_radius_m)
    movel([0.170866, -1.331397, -2.603182, -0.777809, 1.570796, 1.741663],accel_mss,speed_ms,0,blend_radius_m)
    movel([0.169188, -1.331949, -2.602830, -0.777610, 1.570796, 1.739984],accel_mss,speed_ms,0,blend_radius_m)
    movel([0.168129, -1.332259, -2.602632, -0.777498, 1.570796, 1.738925],accel_mss,speed_ms,0,blend_radius_m)
    movel([0.167655, -1.332385, -2.602552, -0.777452, 1.570796, 1.738451],accel_mss,speed_ms,0,blend_radius_m)
    movel([0.167104, -1.332482, -2.602490, -0.777417, 1.570796, 1.737900],accel_mss,speed_ms,0,blend_radius_m)
    movel([0.166831, -1.332495, -2.602481, -0.777412, 1.570796, 1.737628],accel_mss,speed_ms,0,blend_radius_m)
    movel([0.166839, -1.332224, -2.602655, -0.777510, 1.570796, 1.737636],accel_mss,speed_ms,0,blend_radius_m)
    movel([0.180630, -1.327519, -2.605645, -0.779225, 1.570796, 1.751426],accel_mss,speed_ms,0,blend_radius_m)
    movel([0.181557, -1.327233, -2.605826, -0.779330, 1.570796, 1.752353],accel_mss,speed_ms,0,blend_radius_m)
    movel([0.182451, -1.326989, -2.605980, -0.779420, 1.570796, 1.753247],accel_mss,speed_ms,0,blend_radius_m)
    movel([0.182724, -1.327027, -2.605956, -0.779406, 1.570796, 1.753520],accel_mss,speed_ms,0,blend_radius_m)
    movel([0.182667, -1.327269, -2.605803, -0.779316, 1.570796, 1.753464],accel_mss,speed_ms,0,blend_radius_m)
    movel([0.182222, -1.327511, -2.605650, -0.779227, 1.570796, 1.753019],accel_mss,speed_ms,0,blend_radius_m)
    movel([0.181339, -1.327869, -2.605424, -0.779096, 1.570796, 1.752135],accel_mss,speed_ms,0,blend_radius_m)
    movel([0.181339, -1.330766, -2.606757, -0.774866, 1.570796, 1.752135],accel_mss,speed_ms,0,blend_radius_m)
    movel([0.178454, -1.331740, -2.606137, -0.774512, 1.570796, 1.749250],accel_mss,speed_ms,0,blend_radius_m)
    movel([0.173139, -1.333529, -2.604995, -0.773865, 1.570796, 1.743935],accel_mss,speed_ms,0,blend_radius_m)
    movel([0.170866, -1.334287, -2.604510, -0.773592, 1.570796, 1.741663],accel_mss,speed_ms,0,blend_radius_m)
    movel([0.169188, -1.334837, -2.604158, -0.773394, 1.570796, 1.739984],accel_mss,speed_ms,0,blend_radius_m)
    movel([0.168129, -1.335147, -2.603959, -0.773283, 1.570796, 1.738925],accel_mss,speed_ms,0,blend_radius_m)
    movel([0.167655, -1.335272, -2.603879, -0.773238, 1.570796, 1.738451],accel_mss,speed_ms,0,blend_radius_m)
    movel([0.167104, -1.335370, -2.603816, -0.773203, 1.570796, 1.737900],accel_mss,speed_ms,0,blend_radius_m)
    movel([0.166831, -1.335383, -2.603808, -0.773199, 1.570796, 1.737628],accel_mss,speed_ms,0,blend_radius_m)
    movel([0.166839, -1.335112, -2.603981, -0.773296, 1.570796, 1.737636],accel_mss,speed_ms,0,blend_radius_m)
    movel([0.180630, -1.330417, -2.606979, -0.774994, 1.570796, 1.751426],accel_mss,speed_ms,0,blend_radius_m)
    movel([0.181557, -1.330131, -2.607160, -0.775098, 1.570796, 1.752353],accel_mss,speed_ms,0,blend_radius_m)
    movel([0.182451, -1.329888, -2.607315, -0.775187, 1.570796, 1.753247],accel_mss,speed_ms,0,blend_radius_m)
    movel([0.182724, -1.329926, -2.607290, -0.775173, 1.570796, 1.753520],accel_mss,speed_ms,0,blend_radius_m)
    movel([0.182667, -1.330167, -2.607137, -0.775085, 1.570796, 1.753464],accel_mss,speed_ms,0,blend_radius_m)
    movel([0.182222, -1.330409, -2.606984, -0.774996, 1.570796, 1.753019],accel_mss,speed_ms,0,blend_radius_m)
    movel([0.181339, -1.330766, -2.606757, -0.774866, 1.570796, 1.752135],accel_mss,speed_ms,0,blend_radius_m)
    movel([0.181339, -1.297216, -2.590373, -0.824800, 1.570796, 1.752135],accel_mss,speed_ms,0,blend_radius_m)
    speed_ms = 1.000
    movel([0.182651, -1.295149, -2.591622, -0.825618, 1.570796, 1.753447],accel_mss,speed_ms,0,blend_radius_m)
    speed_ms = 0.008
    movel([0.182651, -1.322393, -2.605098, -0.784898, 1.570796, 1.753447],accel_mss,speed_ms,0,blend_radius_m)
    speed_ms = 0.003
    movel([0.182651, -1.325841, -2.606705, -0.779843, 1.570796, 1.753447],accel_mss,speed_ms,0,blend_radius_m)
    speed_ms = 0.008
    movel([0.182368, -1.325922, -2.606654, -0.779813, 1.570796, 1.753165],accel_mss,speed_ms,0,blend_radius_m)
    movel([0.180523, -1.326512, -2.606282, -0.779596, 1.570796, 1.751319],accel_mss,speed_ms,0,blend_radius_m)
    movel([0.173299, -1.328860, -2.604796, -0.778733, 1.570796, 1.744095],accel_mss,speed_ms,0,blend_radius_m)
    movel([0.170475, -1.329768, -2.604219, -0.778401, 1.570796, 1.741271],accel_mss,speed_ms,0,blend_radius_m)
    movel([0.169158, -1.330183, -2.603956, -0.778250, 1.570796, 1.739954],accel_mss,speed_ms,0,blend_radius_m)
    movel([0.167968, -1.330486, -2.603763, -0.778140, 1.570796, 1.738764],accel_mss,speed_ms,0,blend_radius_m)
    movel([0.172335, -1.308218, -2.617604, -0.786567, 1.570796, 1.743131],accel_mss,speed_ms,0,blend_radius_m)
    movel([0.187430, -1.304296, -2.619974, -0.788119, 1.570796, 1.758226],accel_mss,speed_ms,0,blend_radius_m)
    movel([0.184875, -1.316746, -2.612381, -0.783262, 1.570796, 1.755671],accel_mss,speed_ms,0,blend_radius_m)
    movel([0.183824, -1.321768, -2.609260, -0.781361, 1.570796, 1.754620],accel_mss,speed_ms,0,blend_radius_m)
    movel([0.183384, -1.323674, -2.608067, -0.780648, 1.570796, 1.754180],accel_mss,speed_ms,0,blend_radius_m)
    movel([0.182904, -1.325605, -2.606854, -0.779931, 1.570796, 1.753701],accel_mss,speed_ms,0,blend_radius_m)
    movel([0.182651, -1.325841, -2.606705, -0.779843, 1.570796, 1.753447],accel_mss,speed_ms,0,blend_radius_m)
    movel([0.182651, -1.328742, -2.608040, -0.775606, 1.570796, 1.753447],accel_mss,speed_ms,0,blend_radius_m)
    movel([0.182368, -1.328823, -2.607989, -0.775577, 1.570796, 1.753165],accel_mss,speed_ms,0,blend_radius_m)
    movel([0.180523, -1.329411, -2.607617, -0.775361, 1.570796, 1.751319],accel_mss,speed_ms,0,blend_radius_m)
    movel([0.173299, -1.331754, -2.606128, -0.774507, 1.570796, 1.744095],accel_mss,speed_ms,0,blend_radius_m)
    movel([0.170475, -1.332661, -2.605550, -0.774178, 1.570796, 1.741271],accel_mss,speed_ms,0,blend_radius_m)
    movel([0.169158, -1.333075, -2.605285, -0.774028, 1.570796, 1.739954],accel_mss,speed_ms,0,blend_radius_m)
    movel([0.167968, -1.333377, -2.605092, -0.773919, 1.570796, 1.738764],accel_mss,speed_ms,0,blend_radius_m)
    movel([0.172335, -1.311155, -2.618965, -0.782269, 1.570796, 1.743131],accel_mss,speed_ms,0,blend_radius_m)
    movel([0.187430, -1.307240, -2.621341, -0.783808, 1.570796, 1.758226],accel_mss,speed_ms,0,blend_radius_m)
    movel([0.184875, -1.319666, -2.613730, -0.778993, 1.570796, 1.755671],accel_mss,speed_ms,0,blend_radius_m)
    movel([0.183824, -1.324677, -2.610602, -0.777110, 1.570796, 1.754620],accel_mss,speed_ms,0,blend_radius_m)
    movel([0.183384, -1.326579, -2.609406, -0.776403, 1.570796, 1.754180],accel_mss,speed_ms,0,blend_radius_m)
    movel([0.182904, -1.328506, -2.608190, -0.775693, 1.570796, 1.753701],accel_mss,speed_ms,0,blend_radius_m)
    movel([0.182651, -1.328742, -2.608040, -0.775606, 1.570796, 1.753447],accel_mss,speed_ms,0,blend_radius_m)
    movel([0.182651, -1.295149, -2.591622, -0.825618, 1.570796, 1.753447],accel_mss,speed_ms,0,blend_radius_m)
    speed_ms = 1.000
    movel([0.180312, -1.274136, -2.604016, -0.834236, 1.570796, 1.751109],accel_mss,speed_ms,0,blend_radius_m)
    speed_ms = 0.008
    movel([0.180312, -1.301720, -2.617779, -0.792891, 1.570796, 1.751109],accel_mss,speed_ms,0,blend_radius_m)
    speed_ms = 0.003
    movel([0.180312, -1.305215, -2.619421, -0.787753, 1.570796, 1.751109],accel_mss,speed_ms,0,blend_radius_m)
    speed_ms = 0.008
    movel([0.176934, -1.306043, -2.618921, -0.787425, 1.570796, 1.747730],accel_mss,speed_ms,0,blend_radius_m)
    movel([0.174806, -1.306523, -2.618631, -0.787235, 1.570796, 1.745602],accel_mss,speed_ms,0,blend_radius_m)
    movel([0.173179, -1.306865, -2.618424, -0.787100, 1.570796, 1.743975],accel_mss,speed_ms,0,blend_radius_m)
    movel([0.173179, -1.306620, -2.618572, -0.787197, 1.570796, 1.743975],accel_mss,speed_ms,0,blend_radius_m)
    movel([0.175090, -1.306037, -2.618925, -0.787427, 1.570796, 1.745886],accel_mss,speed_ms,0,blend_radius_m)
    movel([0.177117, -1.305471, -2.619266, -0.787651, 1.570796, 1.747913],accel_mss,speed_ms,0,blend_radius_m)
    movel([0.180431, -1.304619, -2.619780, -0.787990, 1.570796, 1.751227],accel_mss,speed_ms,0,blend_radius_m)
    movel([0.183735, -1.303815, -2.620263, -0.788310, 1.570796, 1.754531],accel_mss,speed_ms,0,blend_radius_m)
    movel([0.185742, -1.303371, -2.620530, -0.788488, 1.570796, 1.756538],accel_mss,speed_ms,0,blend_radius_m)
    movel([0.187570, -1.303005, -2.620750, -0.788634, 1.570796, 1.758366],accel_mss,speed_ms,0,blend_radius_m)
    movel([0.187570, -1.303251, -2.620602, -0.788535, 1.570796, 1.758367],accel_mss,speed_ms,0,blend_radius_m)
    movel([0.185853, -1.303760, -2.620296, -0.788332, 1.570796, 1.756649],accel_mss,speed_ms,0,blend_radius_m)
    movel([0.183698, -1.304351, -2.619941, -0.788097, 1.570796, 1.754495],accel_mss,speed_ms,0,blend_radius_m)
    movel([0.180312, -1.305215, -2.619421, -0.787753, 1.570796, 1.751109],accel_mss,speed_ms,0,blend_radius_m)
    movel([0.180312, -1.308157, -2.620786, -0.783446, 1.570796, 1.751109],accel_mss,speed_ms,0,blend_radius_m)
    movel([0.176934, -1.308983, -2.620285, -0.783120, 1.570796, 1.747730],accel_mss,speed_ms,0,blend_radius_m)
    movel([0.174806, -1.309462, -2.619994, -0.782932, 1.570796, 1.745602],accel_mss,speed_ms,0,blend_radius_m)
    movel([0.173179, -1.309804, -2.619787, -0.782798, 1.570796, 1.743975],accel_mss,speed_ms,0,blend_radius_m)
    movel([0.173179, -1.309560, -2.619935, -0.782894, 1.570796, 1.743975],accel_mss,speed_ms,0,blend_radius_m)
    movel([0.175090, -1.308977, -2.620289, -0.783123, 1.570796, 1.745886],accel_mss,speed_ms,0,blend_radius_m)
    movel([0.177117, -1.308413, -2.620631, -0.783345, 1.570796, 1.747913],accel_mss,speed_ms,0,blend_radius_m)
    movel([0.180431, -1.307562, -2.621146, -0.783681, 1.570796, 1.751227],accel_mss,speed_ms,0,blend_radius_m)
    movel([0.183735, -1.306760, -2.621631, -0.783998, 1.570796, 1.754531],accel_mss,speed_ms,0,blend_radius_m)
    movel([0.185742, -1.306317, -2.621898, -0.784174, 1.570796, 1.756538],accel_mss,speed_ms,0,blend_radius_m)
    movel([0.187570, -1.305952, -2.622118, -0.784319, 1.570796, 1.758366],accel_mss,speed_ms,0,blend_radius_m)
    movel([0.187570, -1.306197, -2.621970, -0.784222, 1.570796, 1.758367],accel_mss,speed_ms,0,blend_radius_m)
    movel([0.185853, -1.306705, -2.621664, -0.784020, 1.570796, 1.756649],accel_mss,speed_ms,0,blend_radius_m)
    movel([0.183698, -1.307295, -2.621308, -0.783786, 1.570796, 1.754495],accel_mss,speed_ms,0,blend_radius_m)
    movel([0.180312, -1.308157, -2.620786, -0.783446, 1.570796, 1.751109],accel_mss,speed_ms,0,blend_radius_m)
    movel([0.180312, -1.274136, -2.604016, -0.834236, 1.570796, 1.751109],accel_mss,speed_ms,0,blend_radius_m)
    speed_ms = 1.000
    movel([0.180549, -1.272923, -2.604715, -0.834751, 1.570796, 1.751345],accel_mss,speed_ms,0,blend_radius_m)
    speed_ms = 0.008
    movel([0.180549, -1.300525, -2.618495, -0.793370, 1.570796, 1.751345],accel_mss,speed_ms,0,blend_radius_m)
    speed_ms = 0.003
    movel([0.180549, -1.304023, -2.620139, -0.788228, 1.570796, 1.751345],accel_mss,speed_ms,0,blend_radius_m)
    speed_ms = 0.008
    movel([0.176229, -1.305095, -2.619493, -0.787801, 1.570796, 1.747025],accel_mss,speed_ms,0,blend_radius_m)
    movel([0.175376, -1.305291, -2.619375, -0.787723, 1.570796, 1.746172],accel_mss,speed_ms,0,blend_radius_m)
    movel([0.174532, -1.305466, -2.619270, -0.787654, 1.570796, 1.745328],accel_mss,speed_ms,0,blend_radius_m)
    movel([0.173971, -1.305562, -2.619212, -0.787616, 1.570796, 1.744767],accel_mss,speed_ms,0,blend_radius_m)
    movel([0.173474, -1.305618, -2.619177, -0.787593, 1.570796, 1.744270],accel_mss,speed_ms,0,blend_radius_m)
    movel([0.173334, -1.305409, -2.619304, -0.787676, 1.570796, 1.744130],accel_mss,speed_ms,0,blend_radius_m)
    movel([0.173577, -1.305130, -2.619472, -0.787787, 1.570796, 1.744374],accel_mss,speed_ms,0,blend_radius_m)
    movel([0.174166, -1.304907, -2.619607, -0.787876, 1.570796, 1.744962],accel_mss,speed_ms,0,blend_radius_m)
    movel([0.174782, -1.304702, -2.619730, -0.787957, 1.570796, 1.745578],accel_mss,speed_ms,0,blend_radius_m)
    movel([0.175604, -1.304457, -2.619877, -0.788054, 1.570796, 1.746400],accel_mss,speed_ms,0,blend_radius_m)
    movel([0.176428, -1.304229, -2.620015, -0.788145, 1.570796, 1.747224],accel_mss,speed_ms,0,blend_radius_m)
    movel([0.180727, -1.303127, -2.620677, -0.788585, 1.570796, 1.751523],accel_mss,speed_ms,0,blend_radius_m)
    movel([0.185019, -1.302074, -2.621308, -0.789007, 1.570796, 1.755815],accel_mss,speed_ms,0,blend_radius_m)
    movel([0.185834, -1.301889, -2.621419, -0.789081, 1.570796, 1.756630],accel_mss,speed_ms,0,blend_radius_m)
    movel([0.186644, -1.301727, -2.621516, -0.789146, 1.570796, 1.757440],accel_mss,speed_ms,0,blend_radius_m)
    movel([0.187241, -1.301628, -2.621575, -0.789186, 1.570796, 1.758037],accel_mss,speed_ms,0,blend_radius_m)
    movel([0.187800, -1.301564, -2.621613, -0.789212, 1.570796, 1.758596],accel_mss,speed_ms,0,blend_radius_m)
    movel([0.187953, -1.301745, -2.621505, -0.789139, 1.570796, 1.758749],accel_mss,speed_ms,0,blend_radius_m)
    movel([0.187710, -1.302051, -2.621322, -0.789016, 1.570796, 1.758506],accel_mss,speed_ms,0,blend_radius_m)
    movel([0.187182, -1.302252, -2.621202, -0.788935, 1.570796, 1.757979],accel_mss,speed_ms,0,blend_radius_m)
    movel([0.186600, -1.302442, -2.621087, -0.788859, 1.570796, 1.757397],accel_mss,speed_ms,0,blend_radius_m)
    movel([0.185739, -1.302695, -2.620936, -0.788758, 1.570796, 1.756535],accel_mss,speed_ms,0,blend_radius_m)
    movel([0.184876, -1.302929, -2.620795, -0.788664, 1.570796, 1.755672],accel_mss,speed_ms,0,blend_radius_m)
    movel([0.180549, -1.304023, -2.620139, -0.788228, 1.570796, 1.751345],accel_mss,speed_ms,0,blend_radius_m)
    movel([0.180549, -1.306967, -2.621506, -0.783916, 1.570796, 1.751345],accel_mss,speed_ms,0,blend_radius_m)
    movel([0.176229, -1.308038, -2.620858, -0.783493, 1.570796, 1.747025],accel_mss,speed_ms,0,blend_radius_m)
    movel([0.175376, -1.308233, -2.620740, -0.783416, 1.570796, 1.746172],accel_mss,speed_ms,0,blend_radius_m)
    movel([0.174532, -1.308407, -2.620634, -0.783347, 1.570796, 1.745328],accel_mss,speed_ms,0,blend_radius_m)
    movel([0.173971, -1.308503, -2.620576, -0.783309, 1.570796, 1.744767],accel_mss,speed_ms,0,blend_radius_m)
    movel([0.173474, -1.308559, -2.620542, -0.783287, 1.570796, 1.744270],accel_mss,speed_ms,0,blend_radius_m)
    movel([0.173334, -1.308351, -2.620669, -0.783369, 1.570796, 1.744130],accel_mss,speed_ms,0,blend_radius_m)
    movel([0.173577, -1.308072, -2.620837, -0.783479, 1.570796, 1.744374],accel_mss,speed_ms,0,blend_radius_m)
    movel([0.174166, -1.307849, -2.620972, -0.783567, 1.570796, 1.744962],accel_mss,speed_ms,0,blend_radius_m)
    movel([0.174782, -1.307645, -2.621096, -0.783648, 1.570796, 1.745578],accel_mss,speed_ms,0,blend_radius_m)
    movel([0.175604, -1.307401, -2.621244, -0.783745, 1.570796, 1.746400],accel_mss,speed_ms,0,blend_radius_m)
    movel([0.176428, -1.307173, -2.621381, -0.783835, 1.570796, 1.747224],accel_mss,speed_ms,0,blend_radius_m)
    movel([0.180727, -1.306073, -2.622045, -0.784271, 1.570796, 1.751523],accel_mss,speed_ms,0,blend_radius_m)
    movel([0.185019, -1.305022, -2.622678, -0.784689, 1.570796, 1.755815],accel_mss,speed_ms,0,blend_radius_m)
    movel([0.185834, -1.304838, -2.622789, -0.784762, 1.570796, 1.756630],accel_mss,speed_ms,0,blend_radius_m)
    movel([0.186644, -1.304676, -2.622886, -0.784827, 1.570796, 1.757440],accel_mss,speed_ms,0,blend_radius_m)
    movel([0.187241, -1.304577, -2.622946, -0.784867, 1.570796, 1.758037],accel_mss,speed_ms,0,blend_radius_m)
    movel([0.187800, -1.304513, -2.622984, -0.784892, 1.570796, 1.758596],accel_mss,speed_ms,0,blend_radius_m)
    movel([0.187953, -1.304694, -2.622875, -0.784820, 1.570796, 1.758749],accel_mss,speed_ms,0,blend_radius_m)
    movel([0.187710, -1.304999, -2.622692, -0.784698, 1.570796, 1.758506],accel_mss,speed_ms,0,blend_radius_m)
    movel([0.187182, -1.305200, -2.622571, -0.784618, 1.570796, 1.757979],accel_mss,speed_ms,0,blend_radius_m)
    movel([0.186600, -1.305390, -2.622457, -0.784543, 1.570796, 1.757397],accel_mss,speed_ms,0,blend_radius_m)
    movel([0.185739, -1.305642, -2.622305, -0.784442, 1.570796, 1.756535],accel_mss,speed_ms,0,blend_radius_m)
    movel([0.184876, -1.305876, -2.622164, -0.784349, 1.570796, 1.755672],accel_mss,speed_ms,0,blend_radius_m)
    movel([0.180549, -1.306967, -2.621506, -0.783916, 1.570796, 1.751345],accel_mss,speed_ms,0,blend_radius_m)
    movel([0.180549, -1.272923, -2.604715, -0.834751, 1.570796, 1.751345],accel_mss,speed_ms,0,blend_radius_m)
    speed_ms = 1.000
    movel([0.180846, -1.271403, -2.605588, -0.835398, 1.570796, 1.751642],accel_mss,speed_ms,0,blend_radius_m)
    speed_ms = 0.008
    movel([0.180846, -1.299028, -2.619389, -0.793972, 1.570796, 1.751642],accel_mss,speed_ms,0,blend_radius_m)
    speed_ms = 0.003
    movel([0.180846, -1.302530, -2.621035, -0.788824, 1.570796, 1.751642],accel_mss,speed_ms,0,blend_radius_m)
    speed_ms = 0.008
    movel([0.176518, -1.303606, -2.620389, -0.788394, 1.570796, 1.747315],accel_mss,speed_ms,0,blend_radius_m)
    movel([0.175664, -1.303803, -2.620271, -0.788315, 1.570796, 1.746460],accel_mss,speed_ms,0,blend_radius_m)
    movel([0.174818, -1.303978, -2.620165, -0.788245, 1.570796, 1.745615],accel_mss,speed_ms,0,blend_radius_m)
    movel([0.174256, -1.304075, -2.620107, -0.788207, 1.570796, 1.745053],accel_mss,speed_ms,0,blend_radius_m)
    movel([0.173758, -1.304132, -2.620073, -0.788184, 1.570796, 1.744555],accel_mss,speed_ms,0,blend_radius_m)
    movel([0.173618, -1.303922, -2.620199, -0.788268, 1.570796, 1.744415],accel_mss,speed_ms,0,blend_radius_m)
    movel([0.173863, -1.303642, -2.620367, -0.788379, 1.570796, 1.744659],accel_mss,speed_ms,0,blend_radius_m)
    movel([0.174452, -1.303418, -2.620502, -0.788469, 1.570796, 1.745248],accel_mss,speed_ms,0,blend_radius_m)
    movel([0.175069, -1.303213, -2.620625, -0.788551, 1.570796, 1.745865],accel_mss,speed_ms,0,blend_radius_m)
    movel([0.175893, -1.302967, -2.620773, -0.788649, 1.570796, 1.746689],accel_mss,speed_ms,0,blend_radius_m)
    movel([0.176718, -1.302738, -2.620910, -0.788741, 1.570796, 1.747515],accel_mss,speed_ms,0,blend_radius_m)
    movel([0.181025, -1.301632, -2.621573, -0.789184, 1.570796, 1.751821],accel_mss,speed_ms,0,blend_radius_m)
    movel([0.185323, -1.300575, -2.622205, -0.789610, 1.570796, 1.756120],accel_mss,speed_ms,0,blend_radius_m)
    movel([0.186140, -1.300389, -2.622315, -0.789685, 1.570796, 1.756936],accel_mss,speed_ms,0,blend_radius_m)
    movel([0.186952, -1.300226, -2.622412, -0.789750, 1.570796, 1.757748],accel_mss,speed_ms,0,blend_radius_m)
    movel([0.187550, -1.300126, -2.622472, -0.789791, 1.570796, 1.758346],accel_mss,speed_ms,0,blend_radius_m)
    movel([0.188109, -1.300062, -2.622510, -0.789816, 1.570796, 1.758906],accel_mss,speed_ms,0,blend_radius_m)
    movel([0.188263, -1.300243, -2.622402, -0.789743, 1.570796, 1.759059],accel_mss,speed_ms,0,blend_radius_m)
    movel([0.188019, -1.300551, -2.622219, -0.789619, 1.570796, 1.758815],accel_mss,speed_ms,0,blend_radius_m)
    movel([0.187491, -1.300752, -2.622099, -0.789538, 1.570796, 1.758287],accel_mss,speed_ms,0,blend_radius_m)
    movel([0.186908, -1.300943, -2.621985, -0.789461, 1.570796, 1.757704],accel_mss,speed_ms,0,blend_radius_m)
    movel([0.186045, -1.301196, -2.621833, -0.789359, 1.570796, 1.756841],accel_mss,speed_ms,0,blend_radius_m)
    movel([0.185180, -1.301432, -2.621692, -0.789265, 1.570796, 1.755976],accel_mss,speed_ms,0,blend_radius_m)
    movel([0.180846, -1.302530, -2.621035, -0.788824, 1.570796, 1.751642],accel_mss,speed_ms,0,blend_radius_m)
    movel([0.180846, -1.305477, -2.622404, -0.784508, 1.570796, 1.751642],accel_mss,speed_ms,0,blend_radius_m)
    movel([0.176518, -1.306551, -2.621757, -0.784081, 1.570796, 1.747315],accel_mss,speed_ms,0,blend_radius_m)
    movel([0.175664, -1.306747, -2.621638, -0.784003, 1.570796, 1.746460],accel_mss,speed_ms,0,blend_radius_m)
    movel([0.174818, -1.306923, -2.621532, -0.783934, 1.570796, 1.745615],accel_mss,speed_ms,0,blend_radius_m)
    movel([0.174256, -1.307019, -2.621474, -0.783896, 1.570796, 1.745053],accel_mss,speed_ms,0,blend_radius_m)
    movel([0.173758, -1.307076, -2.621440, -0.783873, 1.570796, 1.744555],accel_mss,speed_ms,0,blend_radius_m)
    movel([0.173618, -1.306867, -2.621566, -0.783956, 1.570796, 1.744415],accel_mss,speed_ms,0,blend_radius_m)
    movel([0.173863, -1.306587, -2.621735, -0.784067, 1.570796, 1.744659],accel_mss,speed_ms,0,blend_radius_m)
    movel([0.174452, -1.306364, -2.621870, -0.784155, 1.570796, 1.745248],accel_mss,speed_ms,0,blend_radius_m)
    movel([0.175069, -1.306159, -2.621993, -0.784237, 1.570796, 1.745865],accel_mss,speed_ms,0,blend_radius_m)
    movel([0.175893, -1.305913, -2.622141, -0.784334, 1.570796, 1.746689],accel_mss,speed_ms,0,blend_radius_m)
    movel([0.176718, -1.305685, -2.622279, -0.784425, 1.570796, 1.747515],accel_mss,speed_ms,0,blend_radius_m)
    movel([0.181025, -1.304581, -2.622943, -0.784865, 1.570796, 1.751821],accel_mss,speed_ms,0,blend_radius_m)
    movel([0.185323, -1.303526, -2.623577, -0.785287, 1.570796, 1.756120],accel_mss,speed_ms,0,blend_radius_m)
    movel([0.186140, -1.303340, -2.623688, -0.785361, 1.570796, 1.756936],accel_mss,speed_ms,0,blend_radius_m)
    movel([0.186952, -1.303178, -2.623785, -0.785426, 1.570796, 1.757748],accel_mss,speed_ms,0,blend_radius_m)
    movel([0.187550, -1.303078, -2.623845, -0.785466, 1.570796, 1.758346],accel_mss,speed_ms,0,blend_radius_m)
    movel([0.188109, -1.303014, -2.623883, -0.785492, 1.570796, 1.758906],accel_mss,speed_ms,0,blend_radius_m)
    movel([0.188263, -1.303195, -2.623775, -0.785419, 1.570796, 1.759059],accel_mss,speed_ms,0,blend_radius_m)
    movel([0.188019, -1.303501, -2.623591, -0.785297, 1.570796, 1.758815],accel_mss,speed_ms,0,blend_radius_m)
    movel([0.187491, -1.303702, -2.623471, -0.785216, 1.570796, 1.758287],accel_mss,speed_ms,0,blend_radius_m)
    movel([0.186908, -1.303893, -2.623356, -0.785140, 1.570796, 1.757704],accel_mss,speed_ms,0,blend_radius_m)
    movel([0.186045, -1.304146, -2.623204, -0.785039, 1.570796, 1.756841],accel_mss,speed_ms,0,blend_radius_m)
    movel([0.185180, -1.304381, -2.623063, -0.784945, 1.570796, 1.755976],accel_mss,speed_ms,0,blend_radius_m)
    movel([0.180846, -1.305477, -2.622404, -0.784508, 1.570796, 1.751642],accel_mss,speed_ms,0,blend_radius_m)
    movel([0.180846, -1.271403, -2.605588, -0.835398, 1.570796, 1.751642],accel_mss,speed_ms,0,blend_radius_m)
    speed_ms = 1.000
    movel([0.180878, -1.269658, -2.606587, -0.836144, 1.570796, 1.751674],accel_mss,speed_ms,0,blend_radius_m)
    speed_ms = 0.008
    movel([0.180878, -1.297310, -2.620412, -0.794668, 1.570796, 1.751674],accel_mss,speed_ms,0,blend_radius_m)
    speed_ms = 0.003
    movel([0.180878, -1.300815, -2.622061, -0.789513, 1.570796, 1.751674],accel_mss,speed_ms,0,blend_radius_m)
    speed_ms = 0.008
    movel([0.173221, -1.302766, -2.620894, -0.788730, 1.570796, 1.744017],accel_mss,speed_ms,0,blend_radius_m)
    movel([0.174123, -1.298088, -2.623685, -0.790616, 1.570796, 1.744920],accel_mss,speed_ms,0,blend_radius_m)
    movel([0.174373, -1.296883, -2.624400, -0.791107, 1.570796, 1.745169],accel_mss,speed_ms,0,blend_radius_m)
    movel([0.174623, -1.295770, -2.625057, -0.791561, 1.570796, 1.745419],accel_mss,speed_ms,0,blend_radius_m)
    movel([0.174967, -1.294373, -2.625881, -0.792134, 1.570796, 1.745763],accel_mss,speed_ms,0,blend_radius_m)
    movel([0.175412, -1.293345, -2.626486, -0.792558, 1.570796, 1.746208],accel_mss,speed_ms,0,blend_radius_m)
    movel([0.190492, -1.289495, -2.628739, -0.794155, 1.570796, 1.761288],accel_mss,speed_ms,0,blend_radius_m)
    movel([0.188541, -1.298906, -2.623199, -0.790284, 1.570796, 1.759338],accel_mss,speed_ms,0,blend_radius_m)
    movel([0.180878, -1.300815, -2.622061, -0.789513, 1.570796, 1.751674],accel_mss,speed_ms,0,blend_radius_m)
    movel([0.180878, -1.303765, -2.623433, -0.785191, 1.570796, 1.751674],accel_mss,speed_ms,0,blend_radius_m)
    movel([0.173221, -1.305712, -2.622262, -0.784414, 1.570796, 1.744017],accel_mss,speed_ms,0,blend_radius_m)
    movel([0.174123, -1.301044, -2.625060, -0.786285, 1.570796, 1.744920],accel_mss,speed_ms,0,blend_radius_m)
    movel([0.174373, -1.299841, -2.625777, -0.786772, 1.570796, 1.745169],accel_mss,speed_ms,0,blend_radius_m)
    movel([0.174623, -1.298730, -2.626436, -0.787222, 1.570796, 1.745419],accel_mss,speed_ms,0,blend_radius_m)
    movel([0.174967, -1.297336, -2.627262, -0.787791, 1.570796, 1.745763],accel_mss,speed_ms,0,blend_radius_m)
    movel([0.175412, -1.296309, -2.627869, -0.788211, 1.570796, 1.746208],accel_mss,speed_ms,0,blend_radius_m)
    movel([0.190492, -1.292466, -2.630127, -0.789796, 1.570796, 1.761288],accel_mss,speed_ms,0,blend_radius_m)
    movel([0.188541, -1.301860, -2.624573, -0.785956, 1.570796, 1.759338],accel_mss,speed_ms,0,blend_radius_m)
    movel([0.180878, -1.303765, -2.623433, -0.785191, 1.570796, 1.751674],accel_mss,speed_ms,0,blend_radius_m)
    movel([0.180878, -1.269658, -2.606587, -0.836144, 1.570796, 1.751674],accel_mss,speed_ms,0,blend_radius_m)
    speed_ms = 1.000
    movel([0.182720, -1.258496, -2.612890, -0.841002, 1.570796, 1.753516],accel_mss,speed_ms,0,blend_radius_m)
    speed_ms = 0.008
